        W2W_1_1_4_2_1_1_1_1 : WSTRING2WSTRING(IN := %opcuaGoodRemoteWrite%);
        W2W_1_1_4_2_1_1_1_1_1 : WSTRING2WSTRING(IN := %opcuaGoodCreateMethod1%);
        W2W_1_1_4_2_1_1_1_1_1_1 : WSTRING2WSTRING(IN := %opcuaGoodCallMethod1%);
        W2W_1_1_4_2_1_1_1_1_1_1_1 : WSTRING2WSTRING(IN := %opcuaGoodSubscribe1%);
        W2W_2 : WSTRING2WSTRING(IN := %opcuaGUIDIdentifier%);
      END_FBS
      SUBAPPLICATION NoSemicolon
        EVENT_INPUT
          REQ;
        END_EVENT
        EVENT_OUTPUT
          CNF;
        END_EVENT
        VAR_INPUT
          ID : ANY_ELEMENTARY;
        END_VAR
      END_SUBAPPLICATION
      SUBAPPLICATION emptyAction
        EVENT_INPUT
          REQ;
        END_EVENT
        EVENT_OUTPUT
          CNF;
        END_EVENT
        VAR_INPUT
          ID : WSTRING;
        END_VAR
      END_SUBAPPLICATION
      SUBAPPLICATION NoExistingAction
        EVENT_INPUT
          REQ;
        END_EVENT
        EVENT_OUTPUT
          CNF;
        END_EVENT
        VAR_INPUT
          ID : WSTRING;
        END_VAR
      END_SUBAPPLICATION
      SUBAPPLICATION UnknownIdentifier
        EVENT_INPUT
          REQ;
        END_EVENT
        EVENT_OUTPUT
          CNF;
        END_EVENT
        VAR_INPUT
          ID : WSTRING;
        END_VAR
      END_SUBAPPLICATION
      SUBAPPLICATION WrongIdentifier
        EVENT_INPUT
          REQ;
        END_EVENT
        EVENT_OUTPUT
          CNF;
        END_EVENT
        VAR_INPUT
          ID : WSTRING;
        END_VAR
      END_SUBAPPLICATION
      SUBAPPLICATION wrongNodeId
        EVENT_INPUT
          REQ;
        END_EVENT
        EVENT_OUTPUT
          CNF;
        END_EVENT
        VAR_INPUT
          ID : WSTRING;
        END_VAR
      END_SUBAPPLICATION
      SUBAPPLICATION wrongPair
        EVENT_INPUT
          REQ;
        END_EVENT
        EVENT_OUTPUT
          CNF;
        END_EVENT
        VAR_INPUT
          ID : WSTRING;
        END_VAR
      END_SUBAPPLICATION
      SUBAPPLICATION LocalWithoutBrowseName
        EVENT_INPUT
          REQ;
        END_EVENT
        EVENT_OUTPUT
          CNF;
        END_EVENT
        VAR_INPUT
          ID : WSTRING;
        END_VAR
      END_SUBAPPLICATION
      SUBAPPLICATION RemoteWithoutBrowseNameNorNodeId
        EVENT_INPUT
          REQ;
        END_EVENT
        EVENT_OUTPUT
          CNF;
        END_EVENT
        VAR_INPUT
          ID : WSTRING;
        END_VAR
      END_SUBAPPLICATION
      SUBAPPLICATION RemoteRead
        EVENT_INPUT
          REQ;
        END_EVENT
        EVENT_OUTPUT
          CNF;
        END_EVENT
        VAR_INPUT
          ID : WSTRING;
        END_VAR
      END_SUBAPPLICATION
      SUBAPPLICATION LocalRead
        EVENT_INPUT
          REQ;
        END_EVENT
        EVENT_OUTPUT
          CNF;
        END_EVENT
        VAR_INPUT
          ID : WSTRING;
        END_VAR
      END_SUBAPPLICATION
      SUBAPPLICATION RemoteWrite
        EVENT_INPUT
          REQ;
        END_EVENT
        EVENT_OUTPUT
          CNF;
        END_EVENT
        VAR_INPUT
          ID : WSTRING;
        END_VAR
      END_SUBAPPLICATION
      SUBAPPLICATION LocalWrite
        EVENT_INPUT
          REQ;
        END_EVENT
        EVENT_OUTPUT
          CNF;
        END_EVENT
        VAR_INPUT
          ID : WSTRING;
        END_VAR
      END_SUBAPPLICATION
      SUBAPPLICATION CreateMethod
        EVENT_INPUT
          REQ;
        END_EVENT
        EVENT_OUTPUT
          CNF;
        END_EVENT
        VAR_INPUT
          ID : WSTRING;
        END_VAR
      END_SUBAPPLICATION
      SUBAPPLICATION CallMethod
        EVENT_INPUT
          REQ;
        END_EVENT
        EVENT_OUTPUT
          CNF;
        END_EVENT
        VAR_INPUT
          ID : WSTRING;
        END_VAR
      END_SUBAPPLICATION
      SUBAPPLICATION Subscribe
        EVENT_INPUT
          REQ;
        END_EVENT
        EVENT_OUTPUT
          CNF;
        END_EVENT
        VAR_INPUT
          ID : WSTRING;
        END_VAR
      END_SUBAPPLICATION
      SUBAPPLICATION GUIDIdentifier
        EVENT_INPUT
          REQ;
        END_EVENT
        EVENT_OUTPUT
          CNF;
        END_EVENT
        VAR_INPUT
          ID : WSTRING;
        END_VAR
      END_SUBAPPLICATION
      EVENT_CONNECTIONS
        NoSemicolon.CNF TO W2W_1.REQ;
        W2W_1.CNF TO emptyAction.REQ;
        emptyAction.CNF TO W2W_1_1.REQ;
        W2W_1_1.CNF TO NoExistingAction.REQ;
        NoExistingAction.CNF TO W2W_1_1_1.REQ;
        UnknownIdentifier.CNF TO W2W_1_1_4.REQ;
        W2W_1_1_4.CNF TO WrongIdentifier.REQ;
        W2W_1_1_3.CNF TO UnknownIdentifier.REQ;
        W2W_1_1_2.CNF TO wrongNodeId.REQ;
        wrongNodeId.CNF TO W2W_1_1_3.REQ;
        W2W_1_1_1.CNF TO wrongPair.REQ;
        wrongPair.CNF TO W2W_1_1_2.REQ;
        W2W.CNF TO NoSemicolon.REQ;
        WrongIdentifier.CNF TO W2W_1_1_4_1.REQ;
        W2W_1_1_4_1.CNF TO LocalWithoutBrowseName.REQ;
        LocalWithoutBrowseName.CNF TO W2W_1_1_4_2.REQ;
        W2W_1_1_4_2.CNF TO RemoteWithoutBrowseNameNorNodeId.REQ;
        W2W_1_1_4_2_1_1.CNF TO RemoteRead.REQ;
        LocalRead.CNF TO W2W_1_1_4_2_1_1.REQ;
        RemoteWithoutBrowseNameNorNodeId.CNF TO W2W_1_1_4_2_1.REQ;
        W2W_1_1_4_2_1.CNF TO LocalRead.REQ;
        RemoteRead.CNF TO W2W_1_1_4_2_1_1_1.REQ;
        W2W_1_1_4_2_1_1_1_1.CNF TO RemoteWrite.REQ;
        W2W_1_1_4_2_1_1_1.CNF TO LocalWrite.REQ;
        LocalWrite.CNF TO W2W_1_1_4_2_1_1_1_1.REQ;
        W2W_1_1_4_2_1_1_1_1_1.CNF TO CreateMethod.REQ;
        RemoteWrite.CNF TO W2W_1_1_4_2_1_1_1_1_1.REQ;
        CreateMethod.CNF TO W2W_1_1_4_2_1_1_1_1_1_1.REQ;
        W2W_1_1_4_2_1_1_1_1_1_1.CNF TO CallMethod.REQ;
        Subscribe.CNF TO STEST_END.REQ;
        CallMethod.CNF TO W2W_1_1_4_2_1_1_1_1_1_1_1.REQ;
        W2W_1_1_4_2_1_1_1_1_1_1_1.CNF TO Subscribe.REQ;
        W2W_2.CNF TO GUIDIdentifier.REQ;
        GUIDIdentifier.CNF TO W2W.REQ;
        START.WARM TO W2W_2.REQ;
        START.COLD TO W2W_2.REQ;
      END_CONNECTIONS
      DATA_CONNECTIONS
        W2W_1_1_4.OUT TO WrongIdentifier.ID;
        W2W_1_1_3.OUT TO UnknownIdentifier.ID;
        W2W_1_1_2.OUT TO wrongNodeId.ID;
        W2W_1_1_1.OUT TO wrongPair.ID;
        W2W_1_1.OUT TO NoExistingAction.ID;
        W2W_1.OUT TO emptyAction.ID;
        W2W.OUT TO NoSemicolon.ID;
        W2W_1_1_4_1.OUT TO LocalWithoutBrowseName.ID;
        W2W_1_1_4_2.OUT TO RemoteWithoutBrowseNameNorNodeId.ID;
        W2W_1_1_4_2_1_1.OUT TO RemoteRead.ID;
        W2W_1_1_4_2_1.OUT TO LocalRead.ID;
        W2W_1_1_4_2_1_1_1_1.OUT TO RemoteWrite.ID;
        W2W_1_1_4_2_1_1_1.OUT TO LocalWrite.ID;
        W2W_1_1_4_2_1_1_1_1_1.OUT TO CreateMethod.ID;
        W2W_1_1_4_2_1_1_1_1_1_1.OUT TO CallMethod.ID;
        W2W_1_1_4_2_1_1_1_1_1_1_1.OUT TO Subscribe.ID;
        W2W_2.OUT TO GUIDIdentifier.ID;
      END_CONNECTIONS
    END_RESOURCE
    RESOURCE foldersReadFirst : EMB_RES
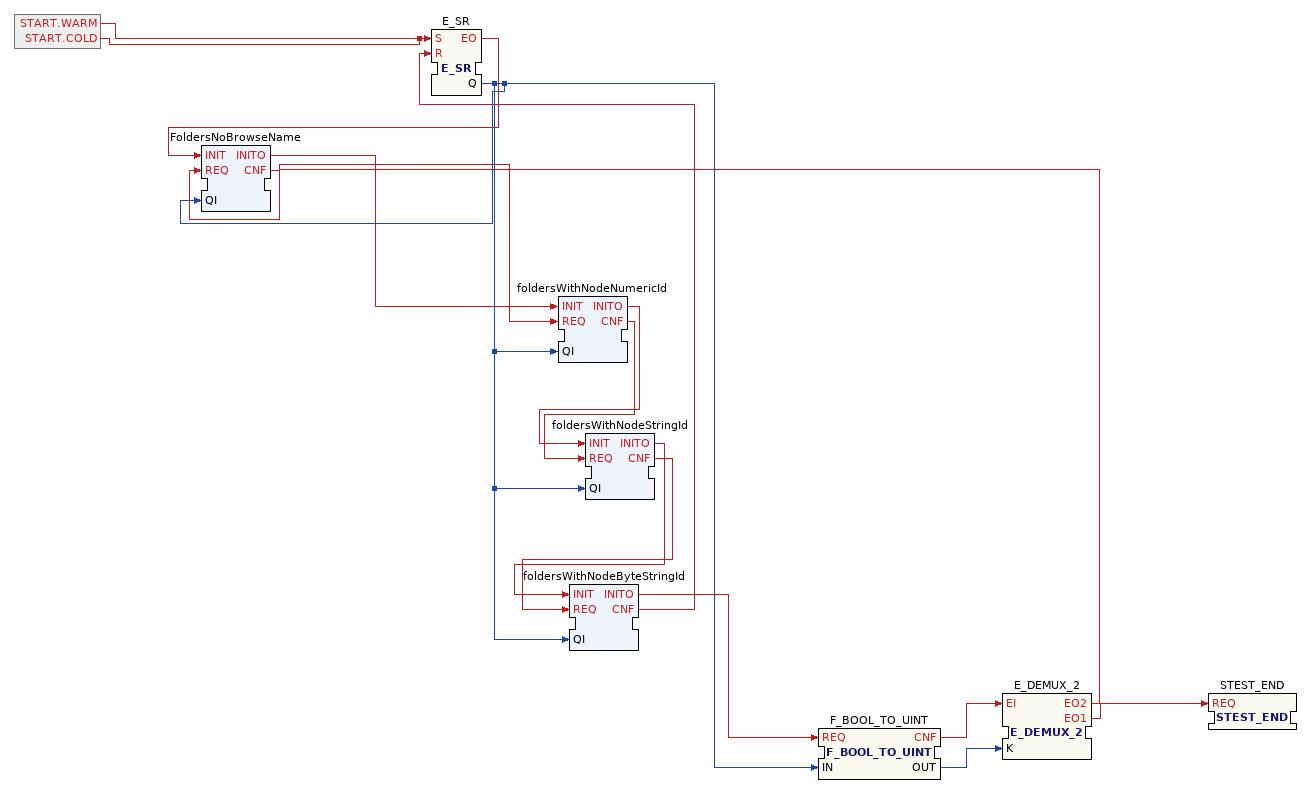
      FBS
        E_SR : E_SR;
        STEST_END : STEST_END;
        E_DEMUX_2 : E_DEMUX_2;
        F_BOOL_TO_UINT : F_BOOL_TO_UINT;
      END_FBS
      SUBAPPLICATION FoldersNoBrowseName
        EVENT_INPUT
          INIT;
          REQ;
        END_EVENT
        EVENT_OUTPUT
          INITO;
          CNF;
        END_EVENT
        VAR_INPUT
          QI : BOOL;
        END_VAR
      END_SUBAPPLICATION
      SUBAPPLICATION foldersWithNodeStringId
        EVENT_INPUT
          INIT;
          REQ;
        END_EVENT
        EVENT_OUTPUT
          INITO;
          CNF;
        END_EVENT
        VAR_INPUT
          QI : BOOL;
        END_VAR
      END_SUBAPPLICATION
      SUBAPPLICATION foldersWithNodeNumericId
        EVENT_INPUT
          INIT;
          REQ;
        END_EVENT
        EVENT_OUTPUT
          INITO;
          CNF;
        END_EVENT
        VAR_INPUT
          QI : BOOL;
        END_VAR
      END_SUBAPPLICATION
      SUBAPPLICATION foldersWithNodeByteStringId
        EVENT_INPUT
          INIT;
          REQ;
        END_EVENT
        EVENT_OUTPUT
          INITO;
          CNF;
        END_EVENT
        VAR_INPUT
          QI : BOOL;
        END_VAR
      END_SUBAPPLICATION
      EVENT_CONNECTIONS
        START.WARM TO E_SR.S;
        START.COLD TO E_SR.S;
        E_SR.EO TO FoldersNoBrowseName.INIT;
        foldersWithNodeStringId.INITO TO foldersWithNodeByteStringId.INIT;
        foldersWithNodeStringId.CNF TO foldersWithNodeByteStringId.REQ;
        E_DEMUX_2.EO2 TO FoldersNoBrowseName.REQ;
        F_BOOL_TO_UINT.CNF TO E_DEMUX_2.EI;
        foldersWithNodeByteStringId.INITO TO F_BOOL_TO_UINT.REQ;
        foldersWithNodeNumericId.CNF TO foldersWithNodeStringId.REQ;
        foldersWithNodeByteStringId.CNF TO E_SR.R;
        foldersWithNodeNumericId.INITO TO foldersWithNodeStringId.INIT;
        FoldersNoBrowseName.INITO TO foldersWithNodeNumericId.INIT;
        FoldersNoBrowseName.CNF TO foldersWithNodeNumericId.REQ;
        E_DEMUX_2.EO1 TO STEST_END.REQ;
      END_CONNECTIONS
      DATA_CONNECTIONS
        E_SR.Q TO FoldersNoBrowseName.QI;
        E_SR.Q TO foldersWithNodeStringId.QI;
        E_SR.Q TO foldersWithNodeNumericId.QI;
        E_SR.Q TO foldersWithNodeByteStringId.QI;
        E_SR.Q TO F_BOOL_TO_UINT.IN;
        F_BOOL_TO_UINT.OUT TO E_DEMUX_2.K;
      END_CONNECTIONS
    END_RESOURCE
    RESOURCE foldersWriteFirst : EMB_RES
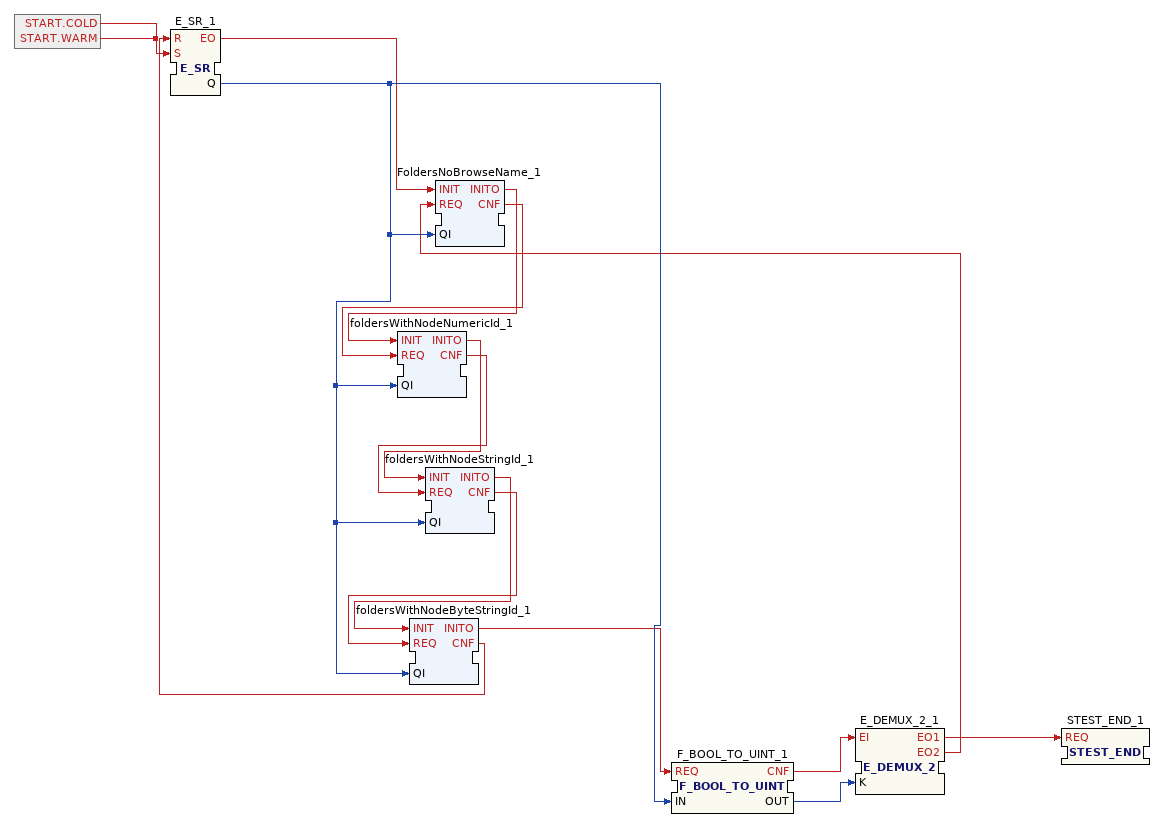
      FBS
        STEST_END_1 : STEST_END;
        F_BOOL_TO_UINT_1 : F_BOOL_TO_UINT;
        E_DEMUX_2_1 : E_DEMUX_2;
        E_SR_1 : E_SR;
      END_FBS
      SUBAPPLICATION FoldersNoBrowseName_1
        EVENT_INPUT
          INIT;
          REQ;
        END_EVENT
        EVENT_OUTPUT
          INITO;
          CNF;
        END_EVENT
        VAR_INPUT
          QI : BOOL;
        END_VAR
      END_SUBAPPLICATION
      SUBAPPLICATION foldersWithNodeByteStringId_1
        EVENT_INPUT
          INIT;
          REQ;
        END_EVENT
        EVENT_OUTPUT
          INITO;
          CNF;
        END_EVENT
        VAR_INPUT
          QI : BOOL;
        END_VAR
      END_SUBAPPLICATION
      SUBAPPLICATION foldersWithNodeNumericId_1
        EVENT_INPUT
          INIT;
          REQ;
        END_EVENT
        EVENT_OUTPUT
          INITO;
          CNF;
        END_EVENT
        VAR_INPUT
          QI : BOOL;
        END_VAR
      END_SUBAPPLICATION
      SUBAPPLICATION foldersWithNodeStringId_1
        EVENT_INPUT
          INIT;
          REQ;
        END_EVENT
        EVENT_OUTPUT
          INITO;
          CNF;
        END_EVENT
        VAR_INPUT
          QI : BOOL;
        END_VAR
      END_SUBAPPLICATION
      EVENT_CONNECTIONS
        FoldersNoBrowseName_1.INITO TO foldersWithNodeNumericId_1.INIT;
        FoldersNoBrowseName_1.CNF TO foldersWithNodeNumericId_1.REQ;
        foldersWithNodeByteStringId_1.INITO TO F_BOOL_TO_UINT_1.REQ;
        foldersWithNodeNumericId_1.INITO TO foldersWithNodeStringId_1.INIT;
        foldersWithNodeNumericId_1.CNF TO foldersWithNodeStringId_1.REQ;
        foldersWithNodeStringId_1.INITO TO foldersWithNodeByteStringId_1.INIT;
        foldersWithNodeStringId_1.CNF TO foldersWithNodeByteStringId_1.REQ;
        F_BOOL_TO_UINT_1.CNF TO E_DEMUX_2_1.EI;
        E_DEMUX_2_1.EO1 TO STEST_END_1.REQ;
        E_DEMUX_2_1.EO2 TO FoldersNoBrowseName_1.REQ;
        foldersWithNodeByteStringId_1.CNF TO E_SR_1.R;
        E_SR_1.EO TO FoldersNoBrowseName_1.INIT;
        START.COLD TO E_SR_1.S;
        START.WARM TO E_SR_1.S;
      END_CONNECTIONS
      DATA_CONNECTIONS
        F_BOOL_TO_UINT_1.OUT TO E_DEMUX_2_1.K;
        E_SR_1.Q TO foldersWithNodeStringId_1.QI;
        E_SR_1.Q TO foldersWithNodeNumericId_1.QI;
        E_SR_1.Q TO FoldersNoBrowseName_1.QI;
        E_SR_1.Q TO foldersWithNodeByteStringId_1.QI;
        E_SR_1.Q TO F_BOOL_TO_UINT_1.IN;
      END_CONNECTIONS
    END_RESOURCE
    RESOURCE createLocalMethods : EMB_RES
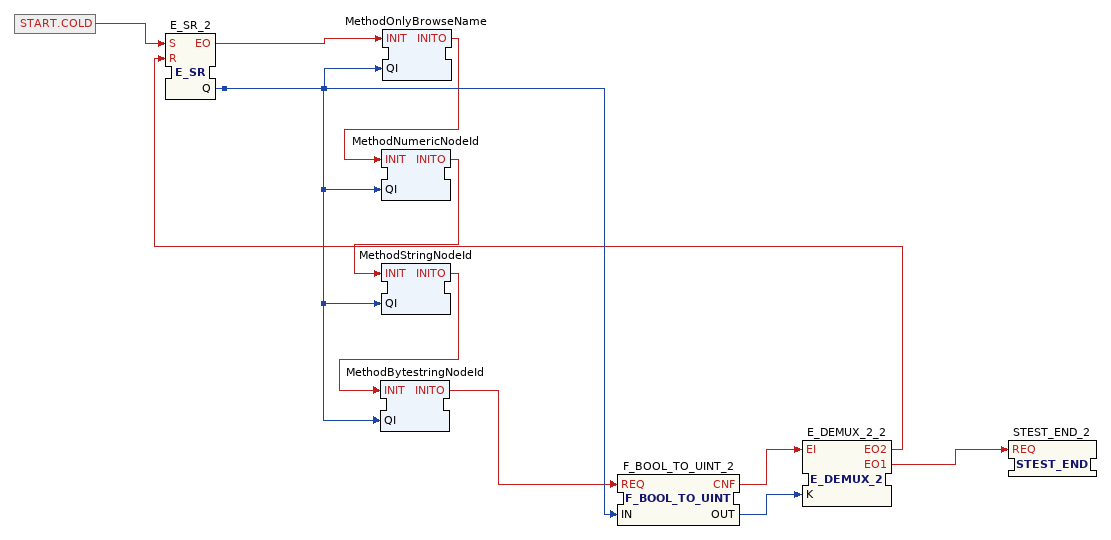
      FBS
        F_BOOL_TO_UINT_2 : F_BOOL_TO_UINT;
        E_DEMUX_2_2 : E_DEMUX_2;
        E_SR_2 : E_SR;
        STEST_END_2 : STEST_END;
      END_FBS
      SUBAPPLICATION MethodOnlyBrowseName
        EVENT_INPUT
          INIT;
        END_EVENT
        EVENT_OUTPUT
          INITO;
        END_EVENT
        VAR_INPUT
          QI : BOOL;
        END_VAR
      END_SUBAPPLICATION
      SUBAPPLICATION MethodBytestringNodeId
        EVENT_INPUT
          INIT;
        END_EVENT
        EVENT_OUTPUT
          INITO;
        END_EVENT
        VAR_INPUT
          QI : BOOL;
        END_VAR
      END_SUBAPPLICATION
      SUBAPPLICATION MethodNumericNodeId
        EVENT_INPUT
          INIT;
        END_EVENT
        EVENT_OUTPUT
          INITO;
        END_EVENT
        VAR_INPUT
          QI : BOOL;
        END_VAR
      END_SUBAPPLICATION
      SUBAPPLICATION MethodStringNodeId
        EVENT_INPUT
          INIT;
        END_EVENT
        EVENT_OUTPUT
          INITO;
        END_EVENT
        VAR_INPUT
          QI : BOOL;
        END_VAR
      END_SUBAPPLICATION
      EVENT_CONNECTIONS
        F_BOOL_TO_UINT_2.CNF TO E_DEMUX_2_2.EI;
        E_SR_2.EO TO MethodOnlyBrowseName.INIT;
        MethodOnlyBrowseName.INITO TO MethodNumericNodeId.INIT;
        MethodNumericNodeId.INITO TO MethodStringNodeId.INIT;
        MethodStringNodeId.INITO TO MethodBytestringNodeId.INIT;
        START.COLD TO E_SR_2.S;
        E_DEMUX_2_2.EO2 TO E_SR_2.R;
        E_DEMUX_2_2.EO1 TO STEST_END_2.REQ;
        MethodBytestringNodeId.INITO TO F_BOOL_TO_UINT_2.REQ;
      END_CONNECTIONS
      DATA_CONNECTIONS
        F_BOOL_TO_UINT_2.OUT TO E_DEMUX_2_2.K;
        E_SR_2.Q TO MethodOnlyBrowseName.QI;
        E_SR_2.Q TO MethodBytestringNodeId.QI;
        E_SR_2.Q TO F_BOOL_TO_UINT_2.IN;
        E_SR_2.Q TO MethodNumericNodeId.QI;
        E_SR_2.Q TO MethodStringNodeId.QI;
      END_CONNECTIONS
    END_RESOURCE
    RESOURCE WorkingServer : EMB_RES
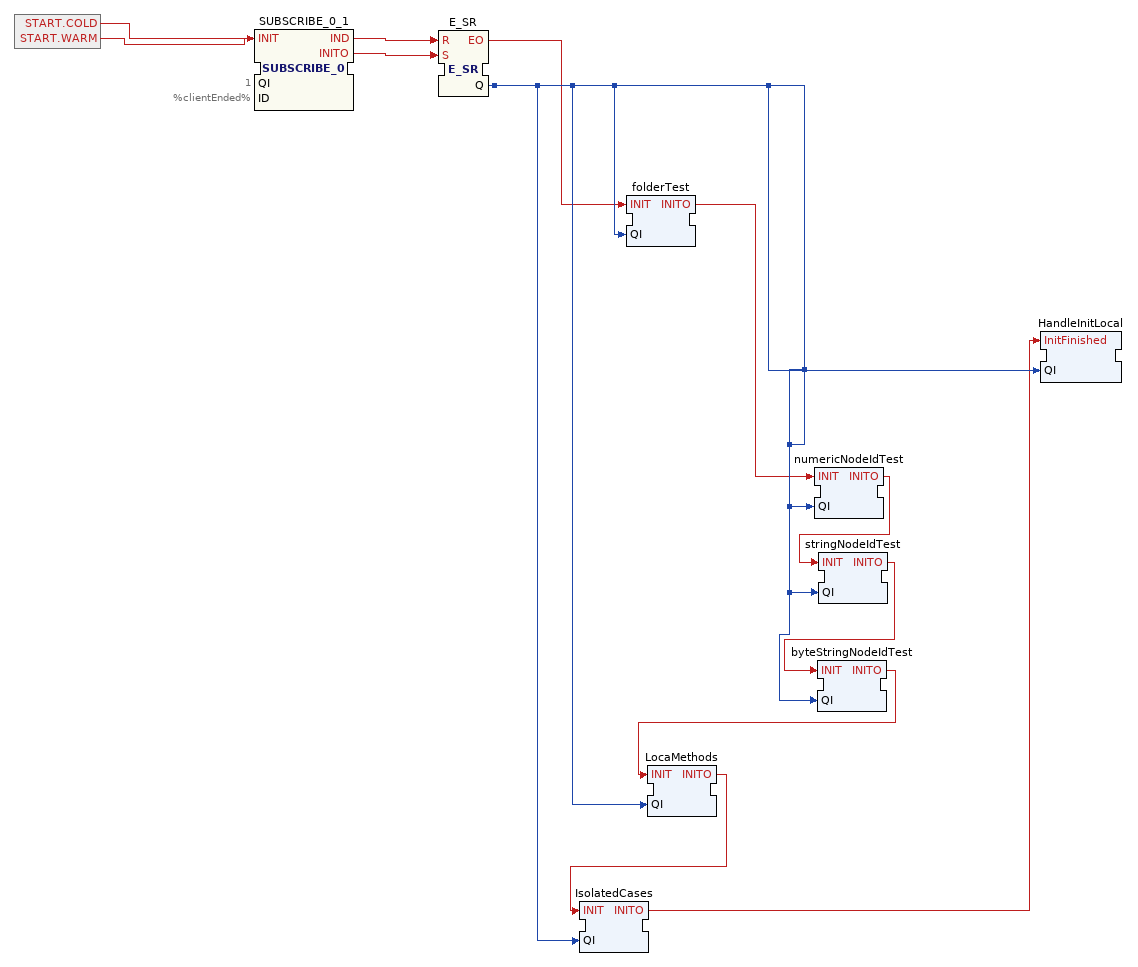
      FBS
        E_SR : E_SR;
        SUBSCRIBE_0_1 : SUBSCRIBE_0(QI := 1, ID := %clientEnded%);
      END_FBS
      SUBAPPLICATION folderTest
        EVENT_INPUT
          INIT;
        END_EVENT
        EVENT_OUTPUT
          INITO;
        END_EVENT
        VAR_INPUT
          QI : BOOL;
        END_VAR
      END_SUBAPPLICATION
      SUBAPPLICATION HandleInitLocal
        EVENT_INPUT
          InitFinished;
        END_EVENT
        VAR_INPUT
          QI : BOOL;
        END_VAR
      END_SUBAPPLICATION
      SUBAPPLICATION LocaMethods
        EVENT_INPUT
          INIT;
        END_EVENT
        EVENT_OUTPUT
          INITO;
        END_EVENT
        VAR_INPUT
          QI : BOOL;
        END_VAR
      END_SUBAPPLICATION
      SUBAPPLICATION stringNodeIdTest
        EVENT_INPUT
          INIT;
        END_EVENT
        EVENT_OUTPUT
          INITO;
        END_EVENT
        VAR_INPUT
          QI : BOOL;
        END_VAR
      END_SUBAPPLICATION
      SUBAPPLICATION byteStringNodeIdTest
        EVENT_INPUT
          INIT;
        END_EVENT
        EVENT_OUTPUT
          INITO;
        END_EVENT
        VAR_INPUT
          QI : BOOL;
        END_VAR
      END_SUBAPPLICATION
      SUBAPPLICATION numericNodeIdTest
        EVENT_INPUT
          INIT;
        END_EVENT
        EVENT_OUTPUT
          INITO;
        END_EVENT
        VAR_INPUT
          QI : BOOL;
        END_VAR
      END_SUBAPPLICATION
      SUBAPPLICATION IsolatedCases
        EVENT_INPUT
          INIT;
        END_EVENT
        EVENT_OUTPUT
          INITO;
        END_EVENT
        VAR_INPUT
          QI : BOOL;
        END_VAR
      END_SUBAPPLICATION
      EVENT_CONNECTIONS
        SUBSCRIBE_0_1.IND TO E_SR.R;
        SUBSCRIBE_0_1.INITO TO E_SR.S;
        START.COLD TO SUBSCRIBE_0_1.INIT;
        START.WARM TO SUBSCRIBE_0_1.INIT;
        E_SR.EO TO folderTest.INIT;
        numericNodeIdTest.INITO TO stringNodeIdTest.INIT;
        stringNodeIdTest.INITO TO byteStringNodeIdTest.INIT;
        byteStringNodeIdTest.INITO TO LocaMethods.INIT;
        folderTest.INITO TO numericNodeIdTest.INIT;
        LocaMethods.INITO TO IsolatedCases.INIT;
        IsolatedCases.INITO TO HandleInitLocal.InitFinished;
      END_CONNECTIONS
      DATA_CONNECTIONS
        E_SR.Q TO folderTest.QI;
        E_SR.Q TO HandleInitLocal.QI;
        E_SR.Q TO numericNodeIdTest.QI;
        E_SR.Q TO stringNodeIdTest.QI;
        E_SR.Q TO byteStringNodeIdTest.QI;
        E_SR.Q TO LocaMethods.QI;
        E_SR.Q TO IsolatedCases.QI;
      END_CONNECTIONS
    END_RESOURCE
    RESOURCE FailingServer : EMB_RES
      FBS
        E_SWITCH : E_SWITCH;
        WorngInputs : TEST_CONDITION(check := 0);
        E_SR : E_SR;
        GoodInputs : TEST_CONDITION;
        SUBSCRIBE_0_1 : SUBSCRIBE_0(QI := 1, ID := %clientEnded%);
        WorngInputsOutputs : TEST_CONDITION(check := 0);
        Writable1 : PUBLISH_1(QI := 1, ID := opc_ua[WRITE;%opcuaFolderTestWithNodeIdNumeric1%/]);
        WorngInputsType : TEST_CONDITION(check := 0);
        BOOL2BOOL_2_1 : DINT2DINT(IN := %opcuaReadValue1%);
        SERVER_0 : SERVER_1(QI := 1, ID := opc_ua[%localMethodAction%;%opcuaMethodCreation5%]);
        SERVER_0_1 : SERVER_1(QI := 1, ID := opc_ua[%localMethodAction%;%opcuaMethodCreation6%]);
        SERVER_0_1_1 : SERVER_1(QI := 1, ID := opc_ua[%localMethodAction%;%opcuaMethodCreation7%]);
        DINT2DINT : DINT2DINT;
        DINT2DINT_1_1 : DINT2DINT;
        DINT2DINT_1 : DINT2DINT;
        SameNodeIdWrite : TEST_CONDITION;
        BOOL2BOOL_2_1_1 : DINT2DINT(IN := %opcuaReadValue1%);
        Writable1_1 : PUBLISH_1(QI := 1, ID := opc_ua[WRITE;/Objects/firstRead/NumericNodeId/folderTests/WithId1,1:i=12345]);
        BOOL2BOOL_2_1_1_1 : DINT2DINT(IN := %opcuaReadValue1%);
        SameNameDifferentNodeIdW : TEST_CONDITION;
        Writable1_1_1 : PUBLISH_1(QI := 1, ID := opc_ua[WRITE;/Objects/firstRead/StringNodeId/folderTests/WithId,1:s=helloWrite]);
        SUBSCRIBE_1_1 : SUBSCRIBE_1(QI := 1, ID := opc_ua[READ;%opcuaFolderTestWithNodeIdNumeric1%]);
        BOOL2BOOL_3_1 : DINT2DINT;
        SUBSCRIBE_1_1_1 : SUBSCRIBE_1(QI := 1, ID := opc_ua[READ;%opcuaFolderTestWithNodeIdNumeric1%]);
        BOOL2BOOL_3 : DINT2DINT;
        SameNodeSecondRead : TEST_CONDITION;
        ReadExistingWritable : TEST_CONDITION;
        F_NOT_1_1 : F_NOT;
        F_NOT : F_NOT;
        SUBSCRIBE_1_1_1_1 : SUBSCRIBE_1(QI := 1, ID := opc_ua[READ;/Objects/firstRead/StringNodeId/folderTests/WithId,1:s=hello]);
        SUBSCRIBE_wrongPath : SUBSCRIBE_1(QI := 1, ID := opc_ua[READ;///]);
        F_NOT_1_2_1_1 : F_NOT;
        SERVER_0_2 : SERVER_1(QI := 1, ID := opc_ua[%localMethodAction%;%opcuaMethodCreation5%]);
        DoubleMethod : TEST_CONDITION;
        BOOL2BOOL_3_2 : DINT2DINT;
        BOOL2BOOL_3_1_1_1 : DINT2DINT;
        F_NOT_1_2_1 : F_NOT;
        ValidNode : TEST_CONDITION;
        WrongPath : TEST_CONDITION;
        BOOL2BOOL_3_1_1 : DINT2DINT;
        BOOL2BOOL_3_2_1_1 : DINT2DINT;
        F_NOT_1_2_1_1_1_1 : F_NOT;
        SUBSCRIBE_150 : SUBSCRIBE_1(QI := 1, ID := opc_ua[READ;%opcuaFolderTestWithNodeIdByteString1%]);
        UnconnectedRD : TEST_CONDITION;
        UnconnectedSD : TEST_CONDITION;
        BOOL2BOOL_3_2_1 : DINT2DINT;
        STRING2STRING_1 : STRING2STRING;
        F_NOT_1 : F_NOT;
        F_NOT_1_2_1_1_1 : F_NOT;
        DifferentTypesOutput : TEST_CONDITION;
        SUBSCRIBE_140 : SUBSCRIBE_2(QI := 1, ID := opc_ua[READ;%opcuaFolderTestWithNodeIdString1%;%opcuaFolderTestWithNodeIdByteString2%]);
        Writable1_1_2 : PUBLISH_2(QI := 1, ID := opc_ua[WRITE;%opcuaFolderTestWithNodeIdString1%;%opcuaFolderTestWithNodeIdByteString2%]);
        SameNodeIdRead : TEST_CONDITION;
        SUBSCRIBE_1 : SUBSCRIBE_1(QI := 1, ID := opc_ua[READ;/Objects/firstRead/NumericNodeId/folderTests/WithId1,1:i=12345]);
        BOOL2BOOL_2_1_1_2 : DINT2DINT;
        F_NOT_2 : F_NOT;
        F_EQ : F_EQ(IN2 := %opcuaReadValue1%);
        SameNameDifferentNodeIdR : TEST_CONDITION;
        Writable1_2 : SUBSCRIBE_1(QI := 1, ID := opc_ua[READ;/Objects/firstRead/StringNodeId/folderTests/WithId,1:s=helloRead]);
        BOOL2BOOL_3_3 : DINT2DINT;
        STRING2STRING : INT2INT;
        BOOL2BOOL_3_2_1_2 : DINT2DINT;
        SameTypesOutput : TEST_CONDITION;
        SUBSCRIBE_150_1 : SUBSCRIBE_1(QI := 1, ID := opc_ua[READ;/Objects/firstRead/StringNodeId/folderTests/WithId,1:s=hello2]);
        F_NOT_1_2_1_2_1 : F_NOT;
        F_NOT_1_2_1_2 : F_NOT;
        BOOL2BOOL_3_1_1_1_1 : DINT2DINT;
        SUBSCRIBE_NoObject_1 : SUBSCRIBE_1(QI := 1, ID := opc_ua[READ;/Objects/firstRead/Methods/1:1:byteStringNodeId/noOParameters]);
        BOOL2BOOL_3_1_1_1_1_1 : DINT2DINT;
        SUBSCRIBE_NoObject : SUBSCRIBE_1(QI := 1, ID := opc_ua[READ;/firstRead/Methods/byteStringNodeId/noOParameters]);
        BrowseWihtouObject : TEST_CONDITION;
        wrongNamespace1 : TEST_CONDITION;
        STRING2STRING_2 : DINT2DINT;
        Timeoutmethod : SERVER_0(QI := 1, ID := opc_ua[%localMethodAction%;%opcuaMethodCreation8%]);
        E_DELAY_1 : E_DELAY(DT := %methodValidDelay%);
        DINT2DINT_1_2 : DINT2DINT(IN := %opcuaReadValue2%);
        PUBLISH_1 : PUBLISH_1(QI := 1, ID := opc_ua[WRITE;%opcuaWRITEVariable%]);
        SERVER_0_3 : SERVER_0(QI := 1, ID := opc_ua[CREATE_METHOD;/Objects]);
        ObjectsFolder : TEST_CONDITION;
        F_NOT_1_2_1_2_1_1 : F_NOT;
        SERVER_0_4 : SERVER_0(QI := 1, ID := opc_ua[CREATE_METHOD;/Objects/notCalledMethod]);
      END_FBS
      SUBAPPLICATION HandleInitLocal
        EVENT_INPUT
          InitFinished;
        END_EVENT
        VAR_INPUT
          QI : BOOL;
        END_VAR
      END_SUBAPPLICATION
      EVENT_CONNECTIONS
        E_SR.EO TO E_SWITCH.EI;
        SUBSCRIBE_0_1.INITO TO E_SR.S;
        SUBSCRIBE_0_1.IND TO E_SR.R;
        E_SWITCH.EO0 TO HandleInitLocal.InitFinished;
        START.COLD TO SUBSCRIBE_0_1.INIT;
        START.WARM TO SUBSCRIBE_0_1.INIT;
        Writable1.CNF TO WorngInputsType.REQ;
        E_SWITCH.EO1 TO SERVER_0.INIT;
        GoodInputs.CNF TO SERVER_0.RSP;
        SERVER_0.INITO TO SERVER_0_1.INIT;
        WorngInputs.CNF TO SERVER_0_1.RSP;
        SERVER_0_1.IND TO WorngInputs.REQ;
        SERVER_0_1.INITO TO SERVER_0_1_1.INIT;
        WorngInputsOutputs.CNF TO SERVER_0_1_1.RSP;
        SERVER_0_1_1.IND TO WorngInputsOutputs.REQ;
        SUBSCRIBE_1_1.INITO TO ReadExistingWritable.REQ;
        ReadExistingWritable.CNF TO SUBSCRIBE_1_1_1.INIT;
        SUBSCRIBE_1_1_1.INITO TO F_NOT_1_1.REQ;
        F_NOT_1_1.CNF TO SameNodeSecondRead.REQ;
        Writable1_1.INITO TO F_NOT.REQ;
        F_NOT.CNF TO SameNodeIdWrite.REQ;
        SERVER_0_2.INITO TO F_NOT_1_2_1_1.REQ;
        F_NOT_1_2_1_1.CNF TO DoubleMethod.REQ;
        SUBSCRIBE_wrongPath.INITO TO F_NOT_1_2_1.REQ;
        F_NOT_1_2_1.CNF TO WrongPath.REQ;
        Writable1_1_1.INITO TO SameNameDifferentNodeIdW.REQ;
        DoubleMethod.CNF TO SUBSCRIBE_150.INIT;
        F_NOT_1.CNF TO UnconnectedSD.REQ;
        SUBSCRIBE_150.INITO TO F_NOT_1_2_1_1_1.REQ;
        F_NOT_1_2_1_1_1.CNF TO DifferentTypesOutput.REQ;
        F_NOT_1_2_1_1_1_1.CNF TO UnconnectedRD.REQ;
        SUBSCRIBE_140.INITO TO F_NOT_1_2_1_1_1_1.REQ;
        UnconnectedRD.CNF TO Writable1_1_2.INIT;
        Writable1_1_2.INITO TO F_NOT_1.REQ;
        SameNodeIdWrite.CNF TO SUBSCRIBE_1.INIT;
        SUBSCRIBE_1.INITO TO F_NOT_2.REQ;
        F_NOT_2.CNF TO SameNodeIdRead.REQ;
        Writable1.INITO TO Writable1_1.INIT;
        SameNodeSecondRead.CNF TO SERVER_0_2.INIT;
        UnconnectedSD.CNF TO SUBSCRIBE_wrongPath.INIT;
        SameNodeIdRead.CNF TO SUBSCRIBE_1_1_1_1.INIT;
        SUBSCRIBE_1_1_1_1.INITO TO Writable1_2.INIT;
        F_EQ.CNF TO ValidNode.REQ;
        SUBSCRIBE_1_1_1_1.IND TO BOOL2BOOL_3_1_1.REQ;
        BOOL2BOOL_3_1_1.CNF TO F_EQ.REQ;
        Writable1_2.INITO TO SameNameDifferentNodeIdR.REQ;
        SameNameDifferentNodeIdR.CNF TO Writable1_1_1.INIT;
        SameNameDifferentNodeIdW.CNF TO SUBSCRIBE_1_1.INIT;
        SameTypesOutput.CNF TO SUBSCRIBE_140.INIT;
        DifferentTypesOutput.CNF TO SUBSCRIBE_150_1.INIT;
        SUBSCRIBE_150_1.INITO TO SameTypesOutput.REQ;
        WrongPath.CNF TO SUBSCRIBE_NoObject.INIT;
        SUBSCRIBE_NoObject.INITO TO F_NOT_1_2_1_2.REQ;
        F_NOT_1_2_1_2.CNF TO BrowseWihtouObject.REQ;
        BrowseWihtouObject.CNF TO SUBSCRIBE_NoObject_1.INIT;
        F_NOT_1_2_1_2_1.CNF TO wrongNamespace1.REQ;
        SUBSCRIBE_NoObject_1.INITO TO F_NOT_1_2_1_2_1.REQ;
        SERVER_0_1_1.INITO TO Timeoutmethod.INIT;
        Timeoutmethod.INITO TO Writable1.INIT;
        SERVER_0.IND TO E_DELAY_1.START;
        E_DELAY_1.EO TO GoodInputs.REQ;
        wrongNamespace1.CNF TO PUBLISH_1.INIT;
        PUBLISH_1.INITO TO SERVER_0_3.INIT;
        SERVER_0_3.INITO TO F_NOT_1_2_1_2_1_1.REQ;
        F_NOT_1_2_1_2_1_1.CNF TO ObjectsFolder.REQ;
        ObjectsFolder.CNF TO SERVER_0_4.INIT;
        SERVER_0_4.INITO TO SERVER_0_4.RSP;
        SERVER_0_4.INITO TO HandleInitLocal.InitFinished;
      END_CONNECTIONS
      DATA_CONNECTIONS
        E_SR.Q TO E_SWITCH.G;
        BOOL2BOOL_2_1.OUT TO Writable1.SD_1;
        SERVER_0.QO TO GoodInputs.check;
        SERVER_0_1_1.RD_1 TO DINT2DINT.IN;
        DINT2DINT.OUT TO SERVER_0_1_1.SD_1;
        SERVER_0.RD_1 TO DINT2DINT_1_1.IN;
        DINT2DINT_1_1.OUT TO SERVER_0.SD_1;
        SERVER_0_1.RD_1 TO DINT2DINT_1.IN;
        DINT2DINT_1.OUT TO SERVER_0_1.SD_1;
        BOOL2BOOL_2_1_1.OUT TO Writable1_1.SD_1;
        BOOL2BOOL_2_1_1_1.OUT TO Writable1_1_1.SD_1;
        SUBSCRIBE_1_1_1.RD_1 TO BOOL2BOOL_3_1.IN;
        SUBSCRIBE_1_1.RD_1 TO BOOL2BOOL_3.IN;
        SUBSCRIBE_1_1.QO TO ReadExistingWritable.check;
        SUBSCRIBE_1_1_1.QO TO F_NOT_1_1.IN;
        F_NOT_1_1.OUT TO SameNodeSecondRead.check;
        Writable1_1.QO TO F_NOT.IN;
        F_NOT.OUT TO SameNodeIdWrite.check;
        SERVER_0_2.QO TO F_NOT_1_2_1_1.IN;
        F_NOT_1_2_1_1.OUT TO DoubleMethod.check;
        SERVER_0_2.RD_1 TO BOOL2BOOL_3_2.IN;
        BOOL2BOOL_3_2.OUT TO SERVER_0_2.SD_1;
        SUBSCRIBE_wrongPath.RD_1 TO BOOL2BOOL_3_1_1_1.IN;
        SUBSCRIBE_wrongPath.QO TO F_NOT_1_2_1.IN;
        F_NOT_1_2_1.OUT TO WrongPath.check;
        SUBSCRIBE_1_1_1_1.RD_1 TO BOOL2BOOL_3_1_1.IN;
        Writable1_1_1.QO TO SameNameDifferentNodeIdW.check;
        SUBSCRIBE_150.RD_1 TO BOOL2BOOL_3_2_1.IN;
        F_NOT_1.OUT TO UnconnectedSD.check;
        SUBSCRIBE_150.QO TO F_NOT_1_2_1_1_1.IN;
        F_NOT_1_2_1_1_1.OUT TO DifferentTypesOutput.check;
        F_NOT_1_2_1_1_1_1.OUT TO UnconnectedRD.check;
        SUBSCRIBE_140.QO TO F_NOT_1_2_1_1_1_1.IN;
        SUBSCRIBE_140.RD_1 TO BOOL2BOOL_3_2_1_1.IN;
        STRING2STRING_1.OUT TO Writable1_1_2.SD_1;
        Writable1_1_2.QO TO F_NOT_1.IN;
        SUBSCRIBE_1.RD_1 TO BOOL2BOOL_2_1_1_2.IN;
        SUBSCRIBE_1.QO TO F_NOT_2.IN;
        F_NOT_2.OUT TO SameNodeIdRead.check;
        F_EQ.OUT TO ValidNode.check;
        BOOL2BOOL_3_1_1.OUT TO F_EQ.IN1;
        Writable1_2.QO TO SameNameDifferentNodeIdR.check;
        Writable1_2.RD_1 TO BOOL2BOOL_3_3.IN;
        SUBSCRIBE_150.RD_1 TO STRING2STRING.IN;
        E_SR.Q TO HandleInitLocal.QI;
        SUBSCRIBE_150_1.RD_1 TO BOOL2BOOL_3_2_1_2.IN;
        SUBSCRIBE_150_1.QO TO SameTypesOutput.check;
        SUBSCRIBE_NoObject_1.QO TO F_NOT_1_2_1_2_1.IN;
        SUBSCRIBE_NoObject_1.RD_1 TO BOOL2BOOL_3_1_1_1_1_1.IN;
        SUBSCRIBE_NoObject.QO TO F_NOT_1_2_1_2.IN;
        SUBSCRIBE_NoObject.RD_1 TO BOOL2BOOL_3_1_1_1_1.IN;
        F_NOT_1_2_1_2.OUT TO BrowseWihtouObject.check;
        F_NOT_1_2_1_2_1.OUT TO wrongNamespace1.check;
        SUBSCRIBE_150_1.RD_1 TO STRING2STRING_2.IN;
        DINT2DINT_1_2.OUT TO PUBLISH_1.SD_1;
        SERVER_0_3.QO TO F_NOT_1_2_1_2_1_1.IN;
        F_NOT_1_2_1_2_1_1.OUT TO ObjectsFolder.check;
      END_CONNECTIONS
    END_RESOURCE
    RESOURCE delayedWorkingServer : EMB_RES
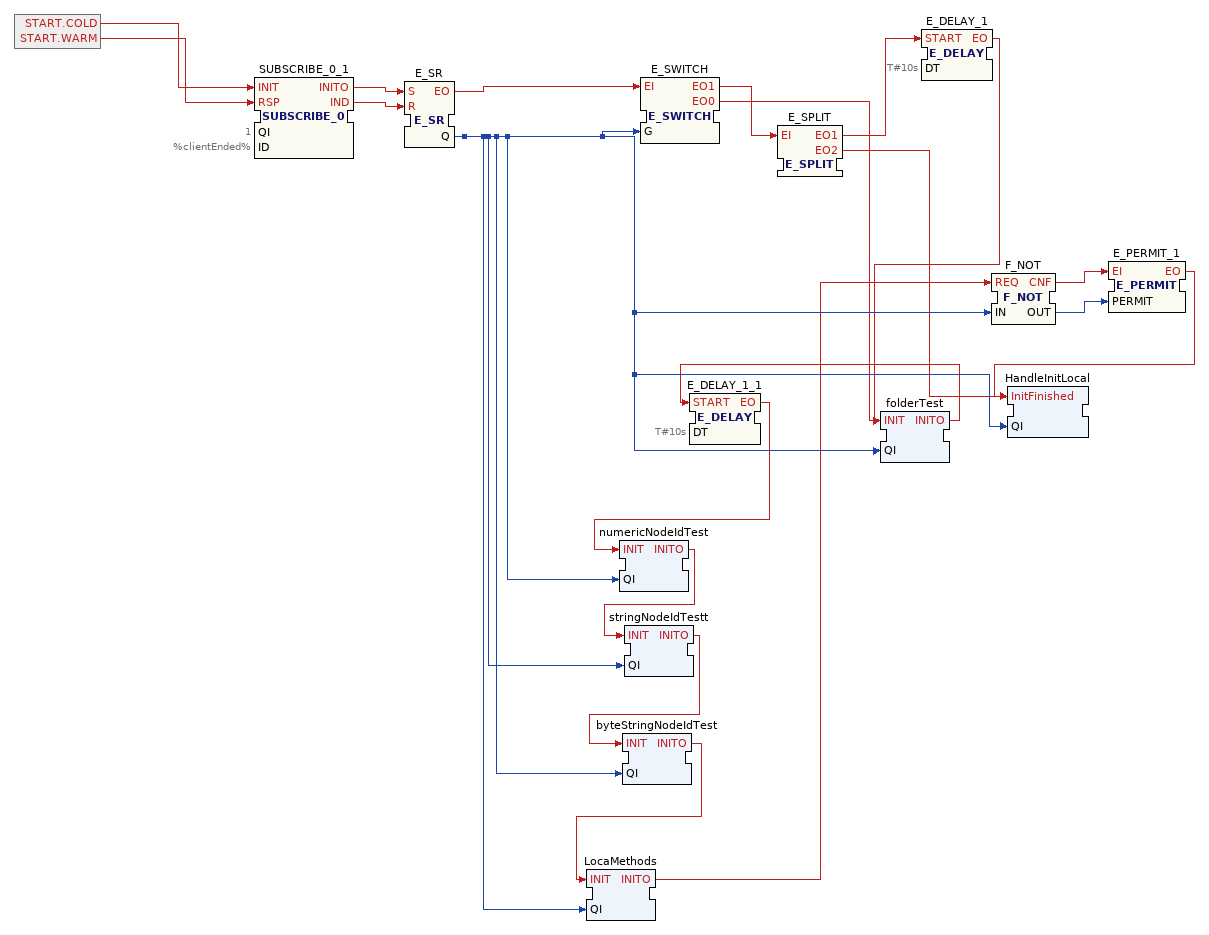
      FBS
        E_SR : E_SR;
        SUBSCRIBE_0_1 : SUBSCRIBE_0(QI := 1, ID := %clientEnded%);
        E_SWITCH : E_SWITCH;
        E_DELAY_1 : E_DELAY(DT := T#10s);
        E_SPLIT : E_SPLIT;
        E_DELAY_1_1 : E_DELAY(DT := T#10s);
        F_NOT : F_NOT;
        E_PERMIT_1 : E_PERMIT;
      END_FBS
      SUBAPPLICATION LocaMethods
        EVENT_INPUT
          INIT;
        END_EVENT
        EVENT_OUTPUT
          INITO;
        END_EVENT
        VAR_INPUT
          QI : BOOL;
        END_VAR
      END_SUBAPPLICATION
      SUBAPPLICATION HandleInitLocal
        EVENT_INPUT
          InitFinished;
        END_EVENT
        VAR_INPUT
          QI : BOOL;
        END_VAR
      END_SUBAPPLICATION
      SUBAPPLICATION numericNodeIdTest
        EVENT_INPUT
          INIT;
        END_EVENT
        EVENT_OUTPUT
          INITO;
        END_EVENT
        VAR_INPUT
          QI : BOOL;
        END_VAR
      END_SUBAPPLICATION
      SUBAPPLICATION folderTest
        EVENT_INPUT
          INIT;
        END_EVENT
        EVENT_OUTPUT
          INITO;
        END_EVENT
        VAR_INPUT
          QI : BOOL;
        END_VAR
      END_SUBAPPLICATION
      SUBAPPLICATION byteStringNodeIdTest
        EVENT_INPUT
          INIT;
        END_EVENT
        EVENT_OUTPUT
          INITO;
        END_EVENT
        VAR_INPUT
          QI : BOOL;
        END_VAR
      END_SUBAPPLICATION
      SUBAPPLICATION stringNodeIdTestt
        EVENT_INPUT
          INIT;
        END_EVENT
        EVENT_OUTPUT
          INITO;
        END_EVENT
        VAR_INPUT
          QI : BOOL;
        END_VAR
      END_SUBAPPLICATION
      EVENT_CONNECTIONS
        SUBSCRIBE_0_1.INITO TO E_SR.S;
        SUBSCRIBE_0_1.IND TO E_SR.R;
        E_SR.EO TO E_SWITCH.EI;
        E_SWITCH.EO1 TO E_SPLIT.EI;
        E_SPLIT.EO1 TO E_DELAY_1.START;
        E_SPLIT.EO2 TO HandleInitLocal.InitFinished;
        LocaMethods.INITO TO F_NOT.REQ;
        F_NOT.CNF TO E_PERMIT_1.EI;
        E_PERMIT_1.EO TO HandleInitLocal.InitFinished;
        START.COLD TO SUBSCRIBE_0_1.INIT;
        START.WARM TO SUBSCRIBE_0_1.RSP;
        numericNodeIdTest.INITO TO stringNodeIdTestt.INIT;
        stringNodeIdTestt.INITO TO byteStringNodeIdTest.INIT;
        folderTest.INITO TO E_DELAY_1_1.START;
        byteStringNodeIdTest.INITO TO LocaMethods.INIT;
        E_SWITCH.EO0 TO folderTest.INIT;
        E_DELAY_1.EO TO folderTest.INIT;
        E_DELAY_1_1.EO TO numericNodeIdTest.INIT;
      END_CONNECTIONS
      DATA_CONNECTIONS
        E_SR.Q TO LocaMethods.QI;
        E_SR.Q TO E_SWITCH.G;
        E_SR.Q TO F_NOT.IN;
        F_NOT.OUT TO E_PERMIT_1.PERMIT;
        E_SR.Q TO HandleInitLocal.QI;
        E_SR.Q TO folderTest.QI;
        E_SR.Q TO stringNodeIdTestt.QI;
        E_SR.Q TO byteStringNodeIdTest.QI;
        E_SR.Q TO numericNodeIdTest.QI;
      END_CONNECTIONS
    END_RESOURCE
    RESOURCE typesServer : EMB_RES
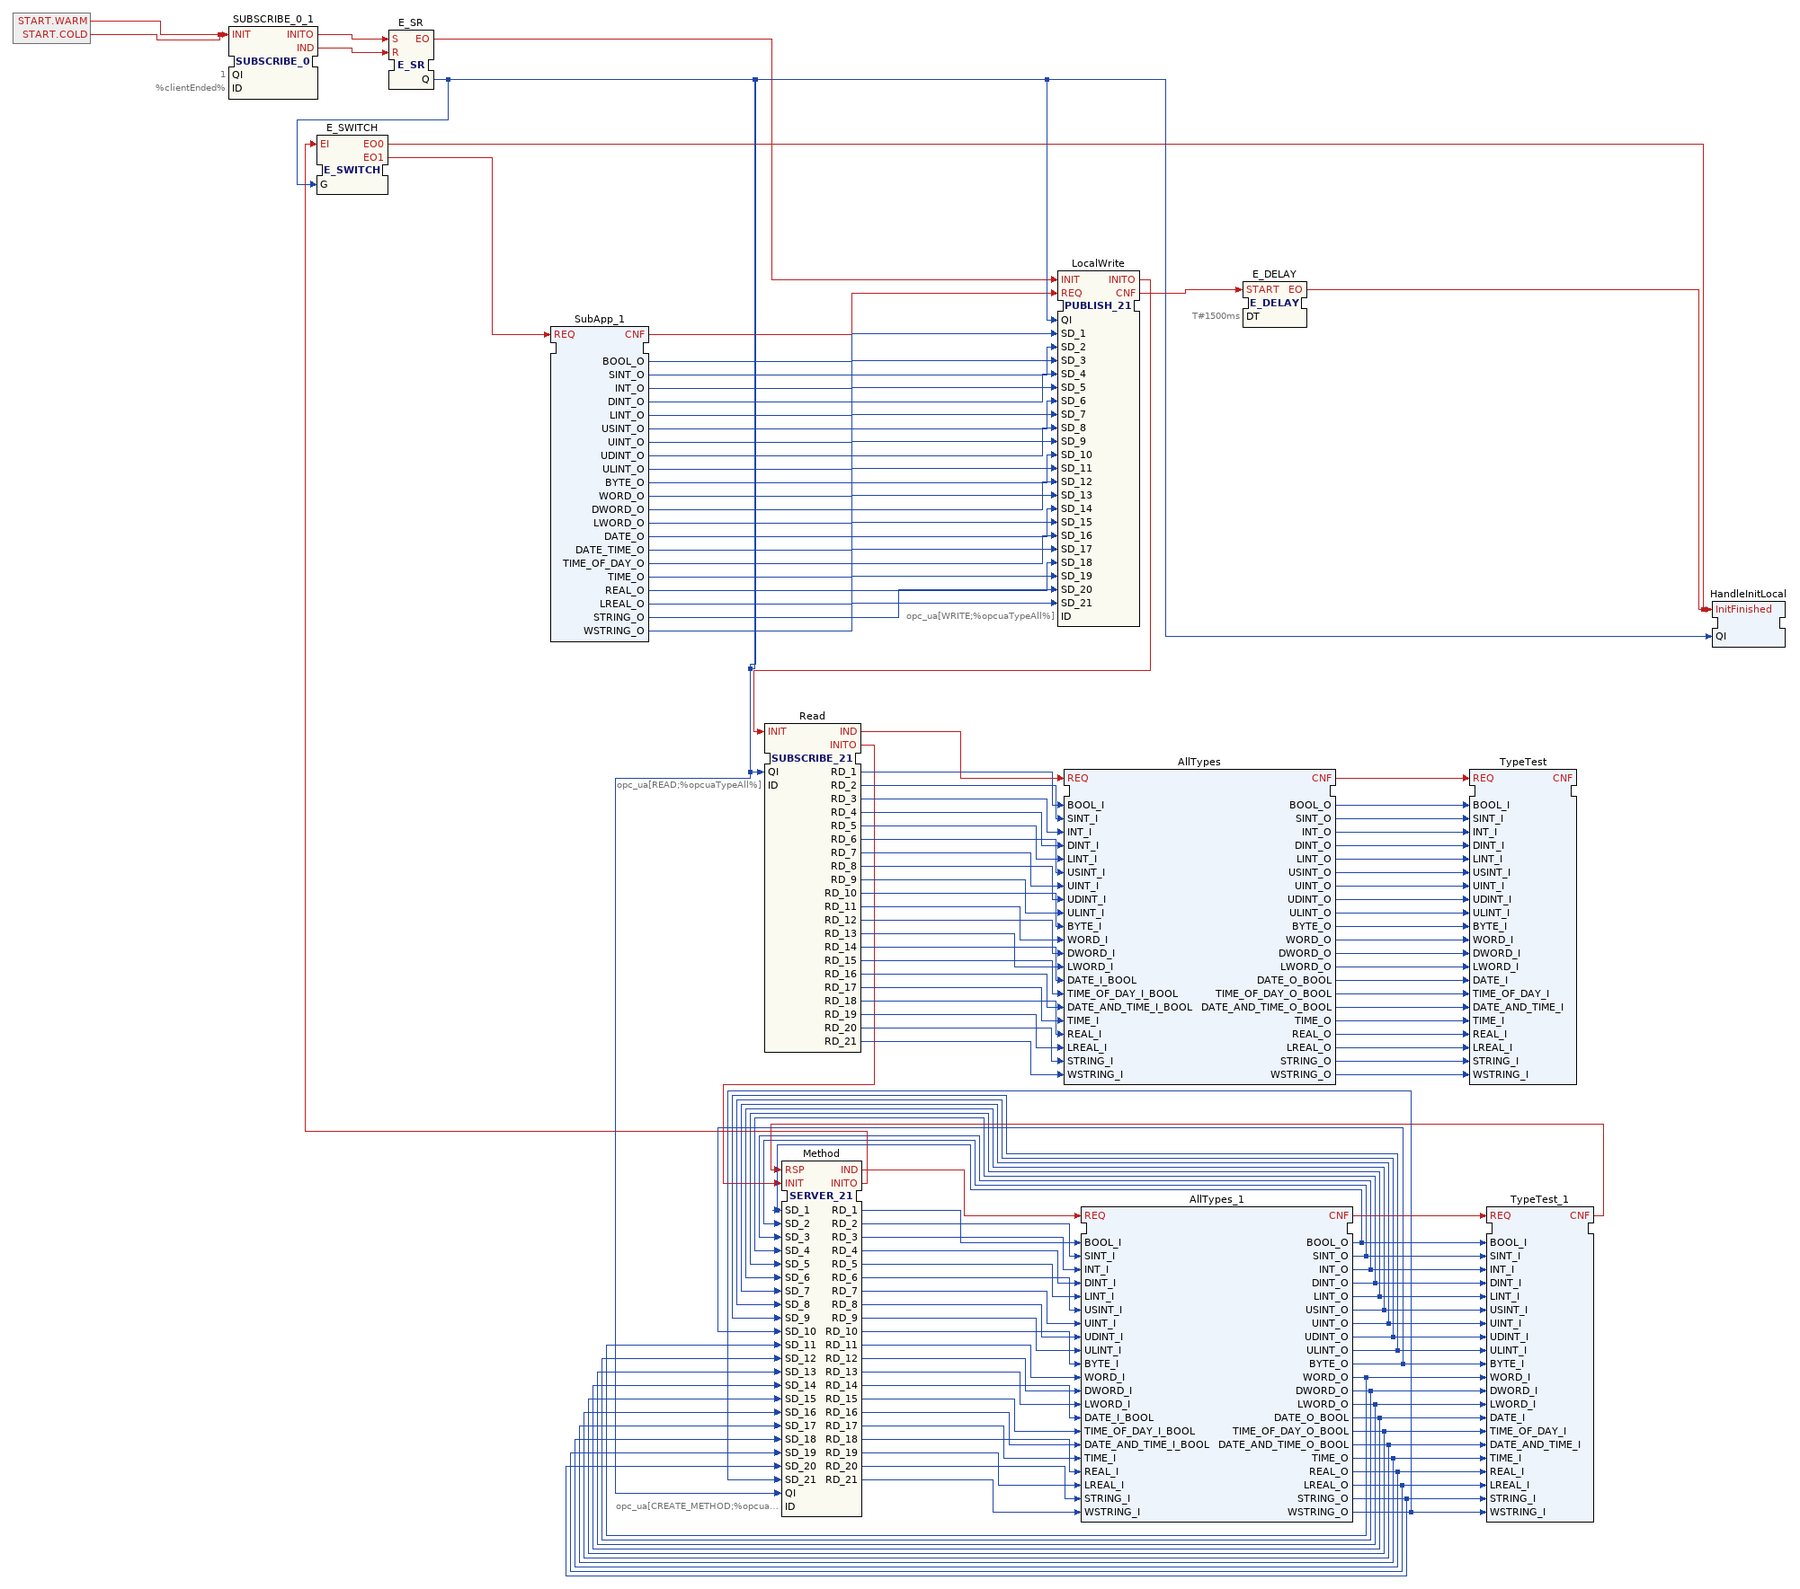
      FBS
        LocalWrite : PUBLISH_21(ID := opc_ua[WRITE;%opcuaTypeAll%]);
        Method : SERVER_21(ID := opc_ua[CREATE_METHOD;%opcuaTypeNode%]);
        Read : SUBSCRIBE_21(ID := opc_ua[READ;%opcuaTypeAll%]);
        E_SR : E_SR;
        SUBSCRIBE_0_1 : SUBSCRIBE_0(QI := 1, ID := %clientEnded%);
        E_SWITCH : E_SWITCH;
        E_DELAY : E_DELAY(DT := T#1500ms);
      END_FBS
      SUBAPPLICATION AllTypes
        EVENT_INPUT
          REQ;
        END_EVENT
        EVENT_OUTPUT
          CNF;
        END_EVENT
        VAR_INPUT
          BOOL_I : BOOL; (* BOOL Type Input *)
          SINT_I : SINT; (* SINT Type Input *)
          INT_I : INT; (* INT Type Input *)
          DINT_I : DINT; (* DINT Type Input *)
          LINT_I : LINT; (* LINT Type Input *)
          USINT_I : USINT; (* USINT Type Input *)
          UINT_I : UINT; (* UINT Type Input *)
          UDINT_I : UDINT; (* UDINT Type Input *)
          ULINT_I : ULINT; (* ULINT Type Input *)
          BYTE_I : BYTE; (* BYTE Type Input *)
          WORD_I : WORD; (* WORD Type Input *)
          DWORD_I : DWORD; (* DWORD Type Input *)
          LWORD_I : LWORD; (* LWORD Type Input *)
          DATE_I_BOOL : BOOL; (* DATE Type Input *)
          TIME_OF_DAY_I_BOOL : BOOL; (* TIME_OF_DAY Type Input *)
          DATE_AND_TIME_I_BOOL : BOOL; (* DATE_AND_TIME Type Input *)
          TIME_I : TIME; (* TIME Type Input *)
          REAL_I : REAL; (* REAL Type Input *)
          LREAL_I : LREAL; (* LREAL Type Input *)
          STRING_I : STRING; (* STRING Type Input *)
          WSTRING_I : WSTRING; (* WSTRING Type Input *)
        END_VAR
        VAR_OUTPUT
          BOOL_O : BOOL; (* BOOL Type Output *)
          SINT_O : SINT; (* SINT Type Output *)
          INT_O : INT; (* INT Type Output *)
          DINT_O : DINT; (* DINT Type Output *)
          LINT_O : LINT; (* LINT Type Output *)
          USINT_O : USINT; (* USINT Type Output *)
          UINT_O : UINT; (* UINT Type Output *)
          UDINT_O : UDINT; (* UDINT Type Output *)
          ULINT_O : ULINT; (* ULINT Type Output *)
          BYTE_O : BYTE; (* BYTE Type Output *)
          WORD_O : WORD; (* WORD Type Output *)
          DWORD_O : DWORD; (* DWORD Type Output *)
          LWORD_O : LWORD; (* LWORD Type Output *)
          DATE_O_BOOL : BOOL; (* DATE Type Output *)
          TIME_OF_DAY_O_BOOL : BOOL; (* TIME_OF_DAY Type Output *)
          DATE_AND_TIME_O_BOOL : BOOL; (* DATE_AND_TIME Type Output *)
          TIME_O : TIME; (* TIME Type Output *)
          REAL_O : REAL; (* REAL Type Output *)
          LREAL_O : LREAL; (* LREAL Type Output *)
          STRING_O : STRING; (* STRING Type Output *)
          WSTRING_O : WSTRING; (* WSTRING Type Output *)
        END_VAR
      END_SUBAPPLICATION
      SUBAPPLICATION TypeTest
        EVENT_INPUT
          REQ;
        END_EVENT
        EVENT_OUTPUT
          CNF;
        END_EVENT
        VAR_INPUT
          BOOL_I : BOOL; (* BOOL Type Input *)
          SINT_I : SINT; (* SINT Type Input *)
          INT_I : INT; (* INT Type Input *)
          DINT_I : DINT; (* DINT Type Input *)
          LINT_I : LINT; (* LINT Type Input *)
          USINT_I : USINT; (* USINT Type Input *)
          UINT_I : UINT; (* UINT Type Input *)
          UDINT_I : UDINT; (* UDINT Type Input *)
          ULINT_I : ULINT; (* ULINT Type Input *)
          BYTE_I : BYTE; (* BYTE Type Input *)
          WORD_I : WORD; (* WORD Type Input *)
          DWORD_I : DWORD; (* DWORD Type Input *)
          LWORD_I : LWORD; (* LWORD Type Input *)
          DATE_I : DATE; (* DATE Type Input *)
          TIME_OF_DAY_I : TIME_OF_DAY; (* TIME_OF_DAY Type Input *)
          DATE_AND_TIME_I : DATE_AND_TIME; (* DATE_AND_TIME Type Input *)
          TIME_I : TIME; (* TIME Type Input *)
          REAL_I : REAL; (* REAL Type Input *)
          LREAL_I : LREAL; (* LREAL Type Input *)
          STRING_I : STRING; (* STRING Type Input *)
          WSTRING_I : WSTRING; (* WSTRING Type Input *)
        END_VAR
      END_SUBAPPLICATION
      SUBAPPLICATION AllTypes_1
        EVENT_INPUT
          REQ;
        END_EVENT
        EVENT_OUTPUT
          CNF;
        END_EVENT
        VAR_INPUT
          BOOL_I : BOOL; (* BOOL Type Input *)
          SINT_I : SINT; (* SINT Type Input *)
          INT_I : INT; (* INT Type Input *)
          DINT_I : DINT; (* DINT Type Input *)
          LINT_I : LINT; (* LINT Type Input *)
          USINT_I : USINT; (* USINT Type Input *)
          UINT_I : UINT; (* UINT Type Input *)
          UDINT_I : UDINT; (* UDINT Type Input *)
          ULINT_I : ULINT; (* ULINT Type Input *)
          BYTE_I : BYTE; (* BYTE Type Input *)
          WORD_I : WORD; (* WORD Type Input *)
          DWORD_I : DWORD; (* DWORD Type Input *)
          LWORD_I : LWORD; (* LWORD Type Input *)
          DATE_I_BOOL : BOOL; (* DATE Type Input *)
          TIME_OF_DAY_I_BOOL : BOOL; (* TIME_OF_DAY Type Input *)
          DATE_AND_TIME_I_BOOL : BOOL; (* DATE_AND_TIME Type Input *)
          TIME_I : TIME; (* TIME Type Input *)
          REAL_I : REAL; (* REAL Type Input *)
          LREAL_I : LREAL; (* LREAL Type Input *)
          STRING_I : STRING; (* STRING Type Input *)
          WSTRING_I : WSTRING; (* WSTRING Type Input *)
        END_VAR
        VAR_OUTPUT
          BOOL_O : BOOL; (* BOOL Type Output *)
          SINT_O : SINT; (* SINT Type Output *)
          INT_O : INT; (* INT Type Output *)
          DINT_O : DINT; (* DINT Type Output *)
          LINT_O : LINT; (* LINT Type Output *)
          USINT_O : USINT; (* USINT Type Output *)
          UINT_O : UINT; (* UINT Type Output *)
          UDINT_O : UDINT; (* UDINT Type Output *)
          ULINT_O : ULINT; (* ULINT Type Output *)
          BYTE_O : BYTE; (* BYTE Type Output *)
          WORD_O : WORD; (* WORD Type Output *)
          DWORD_O : DWORD; (* DWORD Type Output *)
          LWORD_O : LWORD; (* LWORD Type Output *)
          DATE_O_BOOL : BOOL; (* DATE Type Output *)
          TIME_OF_DAY_O_BOOL : BOOL; (* TIME_OF_DAY Type Output *)
          DATE_AND_TIME_O_BOOL : BOOL; (* DATE_AND_TIME Type Output *)
          TIME_O : TIME; (* TIME Type Output *)
          REAL_O : REAL; (* REAL Type Output *)
          LREAL_O : LREAL; (* LREAL Type Output *)
          STRING_O : STRING; (* STRING Type Output *)
          WSTRING_O : WSTRING; (* WSTRING Type Output *)
        END_VAR
      END_SUBAPPLICATION
      SUBAPPLICATION TypeTest_1
        EVENT_INPUT
          REQ;
        END_EVENT
        EVENT_OUTPUT
          CNF;
        END_EVENT
        VAR_INPUT
          BOOL_I : BOOL; (* BOOL Type Input *)
          SINT_I : SINT; (* SINT Type Input *)
          INT_I : INT; (* INT Type Input *)
          DINT_I : DINT; (* DINT Type Input *)
          LINT_I : LINT; (* LINT Type Input *)
          USINT_I : USINT; (* USINT Type Input *)
          UINT_I : UINT; (* UINT Type Input *)
          UDINT_I : UDINT; (* UDINT Type Input *)
          ULINT_I : ULINT; (* ULINT Type Input *)
          BYTE_I : BYTE; (* BYTE Type Input *)
          WORD_I : WORD; (* WORD Type Input *)
          DWORD_I : DWORD; (* DWORD Type Input *)
          LWORD_I : LWORD; (* LWORD Type Input *)
          DATE_I : DATE; (* DATE Type Input *)
          TIME_OF_DAY_I : TIME_OF_DAY; (* TIME_OF_DAY Type Input *)
          DATE_AND_TIME_I : DATE_AND_TIME; (* DATE_AND_TIME Type Input *)
          TIME_I : TIME; (* TIME Type Input *)
          REAL_I : REAL; (* REAL Type Input *)
          LREAL_I : LREAL; (* LREAL Type Input *)
          STRING_I : STRING; (* STRING Type Input *)
          WSTRING_I : WSTRING; (* WSTRING Type Input *)
        END_VAR
      END_SUBAPPLICATION
      SUBAPPLICATION HandleInitLocal
        EVENT_INPUT
          InitFinished;
        END_EVENT
        VAR_INPUT
          QI : BOOL;
        END_VAR
      END_SUBAPPLICATION
      SUBAPPLICATION SubApp_1
        EVENT_INPUT
          REQ;
        END_EVENT
        EVENT_OUTPUT
          CNF;
        END_EVENT
        VAR_OUTPUT
          BOOL_O : BOOL;
          SINT_O : SINT;
          INT_O : INT;
          DINT_O : DINT;
          LINT_O : LINT;
          USINT_O : USINT;
          UINT_O : UINT;
          UDINT_O : UDINT;
          ULINT_O : ULINT;
          BYTE_O : BYTE;
          WORD_O : WORD;
          DWORD_O : DWORD;
          LWORD_O : LWORD;
          DATE_O : BOOL;
          DATE_TIME_O : BOOL;
          TIME_OF_DAY_O : BOOL;
          TIME_O : TIME;
          REAL_O : REAL;
          LREAL_O : LREAL;
          STRING_O : STRING;
          WSTRING_O : WSTRING;
        END_VAR
      END_SUBAPPLICATION
      EVENT_CONNECTIONS
        AllTypes.CNF TO TypeTest.REQ;
        Method.IND TO AllTypes_1.REQ;
        Read.IND TO AllTypes.REQ;
        AllTypes_1.CNF TO TypeTest_1.REQ;
        TypeTest_1.CNF TO Method.RSP;
        SUBSCRIBE_0_1.INITO TO E_SR.S;
        SUBSCRIBE_0_1.IND TO E_SR.R;
        LocalWrite.INITO TO Read.INIT;
        Read.INITO TO Method.INIT;
        START.WARM TO SUBSCRIBE_0_1.INIT;
        START.COLD TO SUBSCRIBE_0_1.INIT;
        E_SR.EO TO LocalWrite.INIT;
        Method.INITO TO E_SWITCH.EI;
        E_SWITCH.EO0 TO HandleInitLocal.InitFinished;
        LocalWrite.CNF TO E_DELAY.START;
        E_DELAY.EO TO HandleInitLocal.InitFinished;
        SubApp_1.CNF TO LocalWrite.REQ;
        E_SWITCH.EO1 TO SubApp_1.REQ;
      END_CONNECTIONS
      DATA_CONNECTIONS
        AllTypes.BOOL_O TO TypeTest.BOOL_I;
        AllTypes.SINT_O TO TypeTest.SINT_I;
        AllTypes.INT_O TO TypeTest.INT_I;
        AllTypes.DINT_O TO TypeTest.DINT_I;
        AllTypes.LINT_O TO TypeTest.LINT_I;
        AllTypes.USINT_O TO TypeTest.USINT_I;
        AllTypes.UINT_O TO TypeTest.UINT_I;
        AllTypes.UDINT_O TO TypeTest.UDINT_I;
        AllTypes.ULINT_O TO TypeTest.ULINT_I;
        AllTypes.BYTE_O TO TypeTest.BYTE_I;
        AllTypes.WORD_O TO TypeTest.WORD_I;
        AllTypes.DWORD_O TO TypeTest.DWORD_I;
        AllTypes.LWORD_O TO TypeTest.LWORD_I;
        AllTypes.DATE_O_BOOL TO TypeTest.DATE_I;
        AllTypes.TIME_OF_DAY_O_BOOL TO TypeTest.TIME_OF_DAY_I;
        AllTypes.DATE_AND_TIME_O_BOOL TO TypeTest.DATE_AND_TIME_I;
        AllTypes.TIME_O TO TypeTest.TIME_I;
        AllTypes.REAL_O TO TypeTest.REAL_I;
        AllTypes.LREAL_O TO TypeTest.LREAL_I;
        AllTypes.STRING_O TO TypeTest.STRING_I;
        AllTypes.WSTRING_O TO TypeTest.WSTRING_I;
        Method.RD_1 TO AllTypes_1.BOOL_I;
        Method.RD_2 TO AllTypes_1.SINT_I;
        Method.RD_3 TO AllTypes_1.INT_I;
        Method.RD_4 TO AllTypes_1.DINT_I;
        Method.RD_5 TO AllTypes_1.LINT_I;
        Method.RD_6 TO AllTypes_1.USINT_I;
        Method.RD_7 TO AllTypes_1.UINT_I;
        Method.RD_8 TO AllTypes_1.UDINT_I;
        Method.RD_9 TO AllTypes_1.ULINT_I;
        Method.RD_10 TO AllTypes_1.BYTE_I;
        Method.RD_11 TO AllTypes_1.WORD_I;
        Method.RD_12 TO AllTypes_1.DWORD_I;
        Method.RD_13 TO AllTypes_1.LWORD_I;
        Method.RD_14 TO AllTypes_1.DATE_I_BOOL;
        Method.RD_15 TO AllTypes_1.TIME_OF_DAY_I_BOOL;
        Method.RD_16 TO AllTypes_1.DATE_AND_TIME_I_BOOL;
        Method.RD_17 TO AllTypes_1.TIME_I;
        Method.RD_18 TO AllTypes_1.REAL_I;
        Method.RD_19 TO AllTypes_1.LREAL_I;
        Method.RD_20 TO AllTypes_1.STRING_I;
        Method.RD_21 TO AllTypes_1.WSTRING_I;
        AllTypes_1.BOOL_O TO Method.SD_1;
        AllTypes_1.SINT_O TO Method.SD_2;
        AllTypes_1.INT_O TO Method.SD_3;
        AllTypes_1.DINT_O TO Method.SD_4;
        AllTypes_1.LINT_O TO Method.SD_5;
        AllTypes_1.USINT_O TO Method.SD_6;
        AllTypes_1.UINT_O TO Method.SD_7;
        AllTypes_1.UDINT_O TO Method.SD_8;
        AllTypes_1.ULINT_O TO Method.SD_9;
        AllTypes_1.BYTE_O TO Method.SD_10;
        AllTypes_1.WORD_O TO Method.SD_11;
        AllTypes_1.DWORD_O TO Method.SD_12;
        AllTypes_1.LWORD_O TO Method.SD_13;
        AllTypes_1.DATE_O_BOOL TO Method.SD_14;
        AllTypes_1.TIME_OF_DAY_O_BOOL TO Method.SD_15;
        AllTypes_1.DATE_AND_TIME_O_BOOL TO Method.SD_16;
        AllTypes_1.TIME_O TO Method.SD_17;
        AllTypes_1.REAL_O TO Method.SD_18;
        AllTypes_1.LREAL_O TO Method.SD_19;
        AllTypes_1.STRING_O TO Method.SD_20;
        AllTypes_1.WSTRING_O TO Method.SD_21;
        Read.RD_1 TO AllTypes.BOOL_I;
        Read.RD_2 TO AllTypes.SINT_I;
        Read.RD_3 TO AllTypes.INT_I;
        Read.RD_4 TO AllTypes.DINT_I;
        Read.RD_5 TO AllTypes.LINT_I;
        Read.RD_6 TO AllTypes.USINT_I;
        Read.RD_7 TO AllTypes.UINT_I;
        Read.RD_8 TO AllTypes.UDINT_I;
        Read.RD_9 TO AllTypes.ULINT_I;
        Read.RD_10 TO AllTypes.BYTE_I;
        Read.RD_11 TO AllTypes.WORD_I;
        Read.RD_12 TO AllTypes.DWORD_I;
        Read.RD_13 TO AllTypes.LWORD_I;
        Read.RD_14 TO AllTypes.DATE_I_BOOL;
        Read.RD_15 TO AllTypes.TIME_OF_DAY_I_BOOL;
        Read.RD_16 TO AllTypes.DATE_AND_TIME_I_BOOL;
        Read.RD_17 TO AllTypes.TIME_I;
        Read.RD_18 TO AllTypes.REAL_I;
        Read.RD_19 TO AllTypes.LREAL_I;
        Read.RD_20 TO AllTypes.STRING_I;
        Read.RD_21 TO AllTypes.WSTRING_I;
        AllTypes_1.BOOL_O TO TypeTest_1.BOOL_I;
        AllTypes_1.SINT_O TO TypeTest_1.SINT_I;
        AllTypes_1.INT_O TO TypeTest_1.INT_I;
        AllTypes_1.DINT_O TO TypeTest_1.DINT_I;
        AllTypes_1.LINT_O TO TypeTest_1.LINT_I;
        AllTypes_1.USINT_O TO TypeTest_1.USINT_I;
        AllTypes_1.UINT_O TO TypeTest_1.UINT_I;
        AllTypes_1.UDINT_O TO TypeTest_1.UDINT_I;
        AllTypes_1.ULINT_O TO TypeTest_1.ULINT_I;
        AllTypes_1.BYTE_O TO TypeTest_1.BYTE_I;
        AllTypes_1.WORD_O TO TypeTest_1.WORD_I;
        AllTypes_1.DWORD_O TO TypeTest_1.DWORD_I;
        AllTypes_1.LWORD_O TO TypeTest_1.LWORD_I;
        AllTypes_1.DATE_O_BOOL TO TypeTest_1.DATE_I;
        AllTypes_1.TIME_OF_DAY_O_BOOL TO TypeTest_1.TIME_OF_DAY_I;
        AllTypes_1.DATE_AND_TIME_O_BOOL TO TypeTest_1.DATE_AND_TIME_I;
        AllTypes_1.TIME_O TO TypeTest_1.TIME_I;
        AllTypes_1.REAL_O TO TypeTest_1.REAL_I;
        AllTypes_1.LREAL_O TO TypeTest_1.LREAL_I;
        AllTypes_1.STRING_O TO TypeTest_1.STRING_I;
        AllTypes_1.WSTRING_O TO TypeTest_1.WSTRING_I;
        E_SR.Q TO HandleInitLocal.QI;
        E_SR.Q TO LocalWrite.QI;
        E_SR.Q TO Read.QI;
        E_SR.Q TO Method.QI;
        E_SR.Q TO E_SWITCH.G;
        SubApp_1.BOOL_O TO LocalWrite.SD_1;
        SubApp_1.SINT_O TO LocalWrite.SD_2;
        SubApp_1.INT_O TO LocalWrite.SD_3;
        SubApp_1.DINT_O TO LocalWrite.SD_4;
        SubApp_1.LINT_O TO LocalWrite.SD_5;
        SubApp_1.USINT_O TO LocalWrite.SD_6;
        SubApp_1.UINT_O TO LocalWrite.SD_7;
        SubApp_1.UDINT_O TO LocalWrite.SD_8;
        SubApp_1.ULINT_O TO LocalWrite.SD_9;
        SubApp_1.BYTE_O TO LocalWrite.SD_10;
        SubApp_1.WORD_O TO LocalWrite.SD_11;
        SubApp_1.DWORD_O TO LocalWrite.SD_12;
        SubApp_1.LWORD_O TO LocalWrite.SD_13;
        SubApp_1.DATE_O TO LocalWrite.SD_14;
        SubApp_1.DATE_TIME_O TO LocalWrite.SD_15;
        SubApp_1.TIME_OF_DAY_O TO LocalWrite.SD_16;
        SubApp_1.TIME_O TO LocalWrite.SD_17;
        SubApp_1.REAL_O TO LocalWrite.SD_18;
        SubApp_1.LREAL_O TO LocalWrite.SD_19;
        SubApp_1.STRING_O TO LocalWrite.SD_20;
        SubApp_1.WSTRING_O TO LocalWrite.SD_21;
      END_CONNECTIONS
    END_RESOURCE
    RESOURCE TestServer : EMB_RES
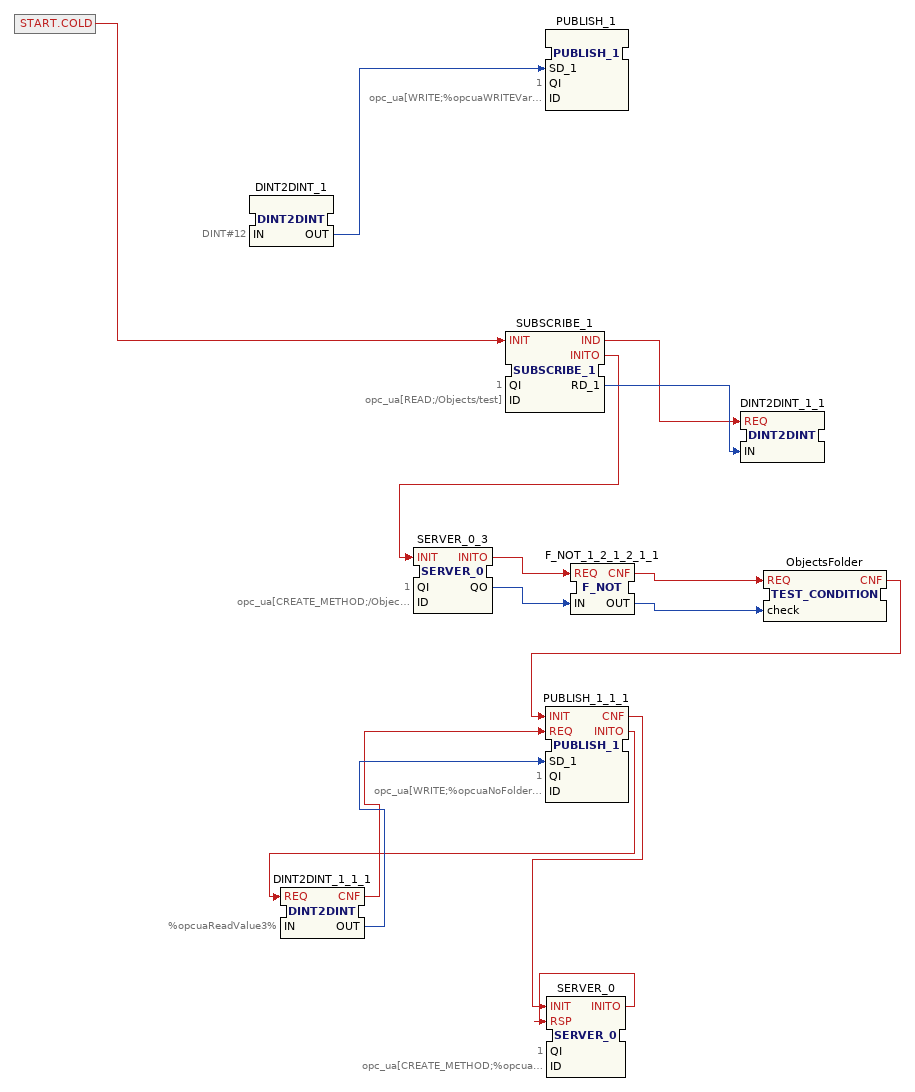
      FBS
        DINT2DINT_1 : DINT2DINT(IN := DINT#12);
        PUBLISH_1 : PUBLISH_1(QI := 1, ID := opc_ua[WRITE;%opcuaWRITEVariable%]);
        SUBSCRIBE_1 : SUBSCRIBE_1(QI := 1, ID := opc_ua[READ;/Objects/test]);
        DINT2DINT_1_1 : DINT2DINT;
        F_NOT_1_2_1_2_1_1 : F_NOT;
        ObjectsFolder : TEST_CONDITION;
        SERVER_0_3 : SERVER_0(QI := 1, ID := opc_ua[CREATE_METHOD;/Objects]);
        PUBLISH_1_1_1 : PUBLISH_1(QI := 1, ID := opc_ua[WRITE;%opcuaNoFolder%]);
        SERVER_0 : SERVER_0(QI := 1, ID := opc_ua[CREATE_METHOD;%opcuaNoFolderMethod%]);
        DINT2DINT_1_1_1 : DINT2DINT(IN := %opcuaReadValue3%);
      END_FBS
      EVENT_CONNECTIONS
        SUBSCRIBE_1.IND TO DINT2DINT_1_1.REQ;
        START.COLD TO SUBSCRIBE_1.INIT;
        F_NOT_1_2_1_2_1_1.CNF TO ObjectsFolder.REQ;
        SERVER_0_3.INITO TO F_NOT_1_2_1_2_1_1.REQ;
        SUBSCRIBE_1.INITO TO SERVER_0_3.INIT;
        ObjectsFolder.CNF TO PUBLISH_1_1_1.INIT;
        PUBLISH_1_1_1.CNF TO SERVER_0.INIT;
        DINT2DINT_1_1_1.CNF TO PUBLISH_1_1_1.REQ;
        SERVER_0.INITO TO SERVER_0.RSP;
        PUBLISH_1_1_1.INITO TO DINT2DINT_1_1_1.REQ;
      END_CONNECTIONS
      DATA_CONNECTIONS
        DINT2DINT_1.OUT TO PUBLISH_1.SD_1;
        SUBSCRIBE_1.RD_1 TO DINT2DINT_1_1.IN;
        F_NOT_1_2_1_2_1_1.OUT TO ObjectsFolder.check;
        SERVER_0_3.QO TO F_NOT_1_2_1_2_1_1.IN;
        DINT2DINT_1_1_1.OUT TO PUBLISH_1_1_1.SD_1;
      END_CONNECTIONS
    END_RESOURCE
  END_DEVICE
  DEVICE OPCUACLient : FORTE_PC(MGR_ID := "localhost:61499")
    {SET_ATTRIBUTE(Profile, HOLOBLOC)} (* device profile *)
    RESOURCE WorkingClient : EMB_RES
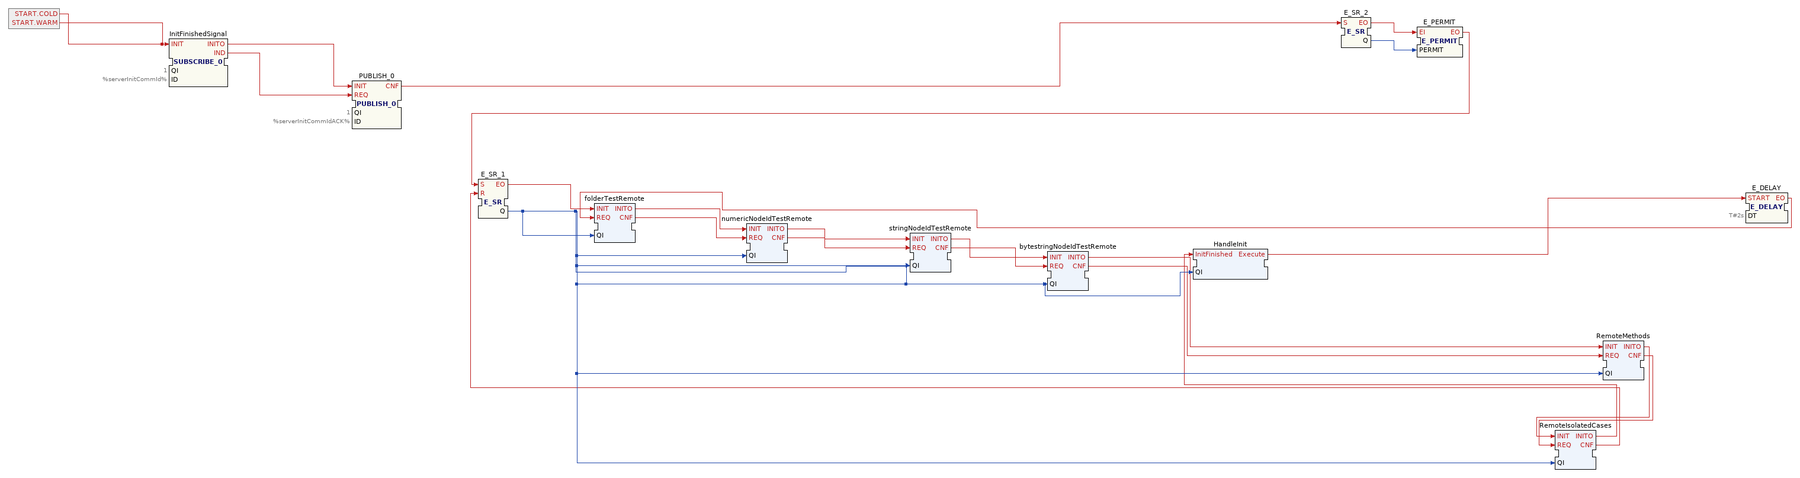
      FBS
        E_SR_1 : E_SR;
        InitFinishedSignal : SUBSCRIBE_0(QI := 1, ID := %serverInitCommId%);
        PUBLISH_0 : PUBLISH_0(QI := 1, ID := %serverInitCommIdACK%);
        E_SR_2 : E_SR;
        E_PERMIT : E_PERMIT;
        E_DELAY : E_DELAY(DT := T#2s);
      END_FBS
      SUBAPPLICATION folderTestRemote
        EVENT_INPUT
          INIT;
          REQ;
        END_EVENT
        EVENT_OUTPUT
          INITO;
          CNF;
        END_EVENT
        VAR_INPUT
          QI : BOOL;
        END_VAR
      END_SUBAPPLICATION
      SUBAPPLICATION HandleInit
        EVENT_INPUT
          InitFinished;
        END_EVENT
        EVENT_OUTPUT
          Execute;
        END_EVENT
        VAR_INPUT
          QI : BOOL;
        END_VAR
      END_SUBAPPLICATION
      SUBAPPLICATION numericNodeIdTestRemote
        EVENT_INPUT
          INIT;
          REQ;
        END_EVENT
        EVENT_OUTPUT
          INITO;
          CNF;
        END_EVENT
        VAR_INPUT
          QI : BOOL;
        END_VAR
      END_SUBAPPLICATION
      SUBAPPLICATION stringNodeIdTestRemote
        EVENT_INPUT
          INIT;
          REQ;
        END_EVENT
        EVENT_OUTPUT
          INITO;
          CNF;
        END_EVENT
        VAR_INPUT
          QI : BOOL;
        END_VAR
      END_SUBAPPLICATION
      SUBAPPLICATION bytestringNodeIdTestRemote
        EVENT_INPUT
          INIT;
          REQ;
        END_EVENT
        EVENT_OUTPUT
          INITO;
          CNF;
        END_EVENT
        VAR_INPUT
          QI : BOOL;
        END_VAR
      END_SUBAPPLICATION
      SUBAPPLICATION RemoteMethods
        EVENT_INPUT
          INIT;
          REQ;
        END_EVENT
        EVENT_OUTPUT
          INITO;
          CNF;
        END_EVENT
        VAR_INPUT
          QI : BOOL;
        END_VAR
      END_SUBAPPLICATION
      SUBAPPLICATION RemoteIsolatedCases
        EVENT_INPUT
          INIT;
          REQ;
        END_EVENT
        EVENT_OUTPUT
          INITO;
          CNF;
        END_EVENT
        VAR_INPUT
          QI : BOOL;
        END_VAR
      END_SUBAPPLICATION
      EVENT_CONNECTIONS
        START.COLD TO InitFinishedSignal.INIT;
        START.WARM TO InitFinishedSignal.INIT;
        InitFinishedSignal.INITO TO PUBLISH_0.INIT;
        folderTestRemote.INITO TO numericNodeIdTestRemote.INIT;
        numericNodeIdTestRemote.INITO TO stringNodeIdTestRemote.INIT;
        stringNodeIdTestRemote.INITO TO bytestringNodeIdTestRemote.INIT;
        InitFinishedSignal.IND TO PUBLISH_0.REQ;
        PUBLISH_0.CNF TO E_SR_2.S;
        E_SR_2.EO TO E_PERMIT.EI;
        E_PERMIT.EO TO E_SR_1.S;
        E_DELAY.EO TO folderTestRemote.REQ;
        HandleInit.Execute TO E_DELAY.START;
        bytestringNodeIdTestRemote.INITO TO RemoteMethods.INIT;
        E_SR_1.EO TO folderTestRemote.INIT;
        bytestringNodeIdTestRemote.CNF TO RemoteMethods.REQ;
        stringNodeIdTestRemote.CNF TO bytestringNodeIdTestRemote.REQ;
        numericNodeIdTestRemote.CNF TO stringNodeIdTestRemote.REQ;
        folderTestRemote.CNF TO numericNodeIdTestRemote.REQ;
        RemoteIsolatedCases.INITO TO HandleInit.InitFinished;
        RemoteMethods.INITO TO RemoteIsolatedCases.INIT;
        RemoteIsolatedCases.CNF TO E_SR_1.R;
        RemoteMethods.CNF TO RemoteIsolatedCases.REQ;
      END_CONNECTIONS
      DATA_CONNECTIONS
        E_SR_1.Q TO folderTestRemote.QI;
        E_SR_1.Q TO HandleInit.QI;
        E_SR_1.Q TO numericNodeIdTestRemote.QI;
        E_SR_1.Q TO stringNodeIdTestRemote.QI;
        E_SR_1.Q TO bytestringNodeIdTestRemote.QI;
        E_SR_2.Q TO E_PERMIT.PERMIT;
        E_SR_1.Q TO RemoteMethods.QI;
        E_SR_1.Q TO RemoteIsolatedCases.QI;
      END_CONNECTIONS
    END_RESOURCE
    RESOURCE WokingClientWithoutSubs : EMB_RES
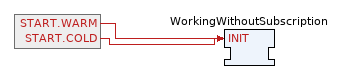
      SUBAPPLICATION WorkingWithoutSubscription
        EVENT_INPUT
          INIT;
        END_EVENT
      END_SUBAPPLICATION
      EVENT_CONNECTIONS
        START.WARM TO WorkingWithoutSubscription.INIT;
        START.COLD TO WorkingWithoutSubscription.INIT;
      END_CONNECTIONS
    END_RESOURCE
    RESOURCE FailingClient : EMB_RES
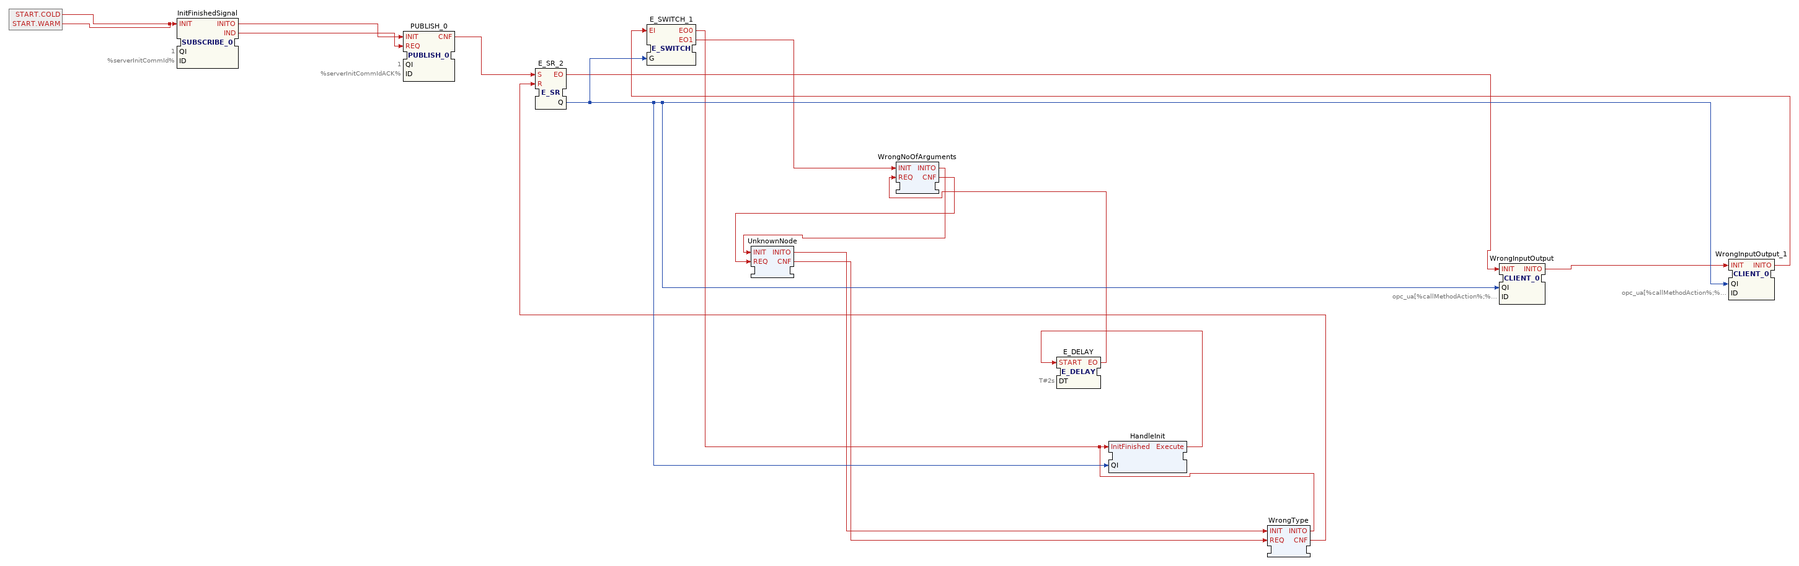
      FBS
        E_SWITCH_1 : E_SWITCH;
        InitFinishedSignal : SUBSCRIBE_0(QI := 1, ID := %serverInitCommId%);
        E_DELAY : E_DELAY(DT := T#2s);
        E_SR_2 : E_SR;
        PUBLISH_0 : PUBLISH_0(QI := 1, ID := %serverInitCommIdACK%);
        WrongInputOutput : CLIENT_0(ID := opc_ua[%callMethodAction%;%unknownEndpoint%;%opcuaMethodCreation7%]);
        WrongInputOutput_1 : CLIENT_0(ID := opc_ua[%callMethodAction%;%unknownEndpoint%;%opcuaMethodCreation7%]);
      END_FBS
      SUBAPPLICATION HandleInit
        EVENT_INPUT
          InitFinished;
        END_EVENT
        EVENT_OUTPUT
          Execute;
        END_EVENT
        VAR_INPUT
          QI : BOOL;
        END_VAR
      END_SUBAPPLICATION
      SUBAPPLICATION UnknownNode
        EVENT_INPUT
          INIT;
          REQ;
        END_EVENT
        EVENT_OUTPUT
          INITO;
          CNF;
        END_EVENT
      END_SUBAPPLICATION
      SUBAPPLICATION WrongNoOfArguments
        EVENT_INPUT
          INIT;
          REQ;
        END_EVENT
        EVENT_OUTPUT
          INITO;
          CNF;
        END_EVENT
      END_SUBAPPLICATION
      SUBAPPLICATION WrongType
        EVENT_INPUT
          INIT;
          REQ;
        END_EVENT
        EVENT_OUTPUT
          INITO;
          CNF;
        END_EVENT
      END_SUBAPPLICATION
      EVENT_CONNECTIONS
        E_SWITCH_1.EO0 TO HandleInit.InitFinished;
        HandleInit.Execute TO E_DELAY.START;
        InitFinishedSignal.INITO TO PUBLISH_0.INIT;
        InitFinishedSignal.IND TO PUBLISH_0.REQ;
        PUBLISH_0.CNF TO E_SR_2.S;
        START.COLD TO InitFinishedSignal.INIT;
        START.WARM TO InitFinishedSignal.INIT;
        E_DELAY.EO TO WrongNoOfArguments.REQ;
        WrongNoOfArguments.CNF TO UnknownNode.REQ;
        WrongNoOfArguments.INITO TO UnknownNode.INIT;
        UnknownNode.INITO TO WrongType.INIT;
        UnknownNode.CNF TO WrongType.REQ;
        WrongType.INITO TO HandleInit.InitFinished;
        WrongType.CNF TO E_SR_2.R;
        WrongInputOutput.INITO TO WrongInputOutput_1.INIT;
        E_SR_2.EO TO WrongInputOutput.INIT;
        E_SWITCH_1.EO1 TO WrongNoOfArguments.INIT;
        WrongInputOutput_1.INITO TO E_SWITCH_1.EI;
      END_CONNECTIONS
      DATA_CONNECTIONS
        E_SR_2.Q TO HandleInit.QI;
        E_SR_2.Q TO E_SWITCH_1.G;
        E_SR_2.Q TO WrongInputOutput.QI;
        E_SR_2.Q TO WrongInputOutput_1.QI;
      END_CONNECTIONS
    END_RESOURCE
    RESOURCE delayedWorkingClient : EMB_RES
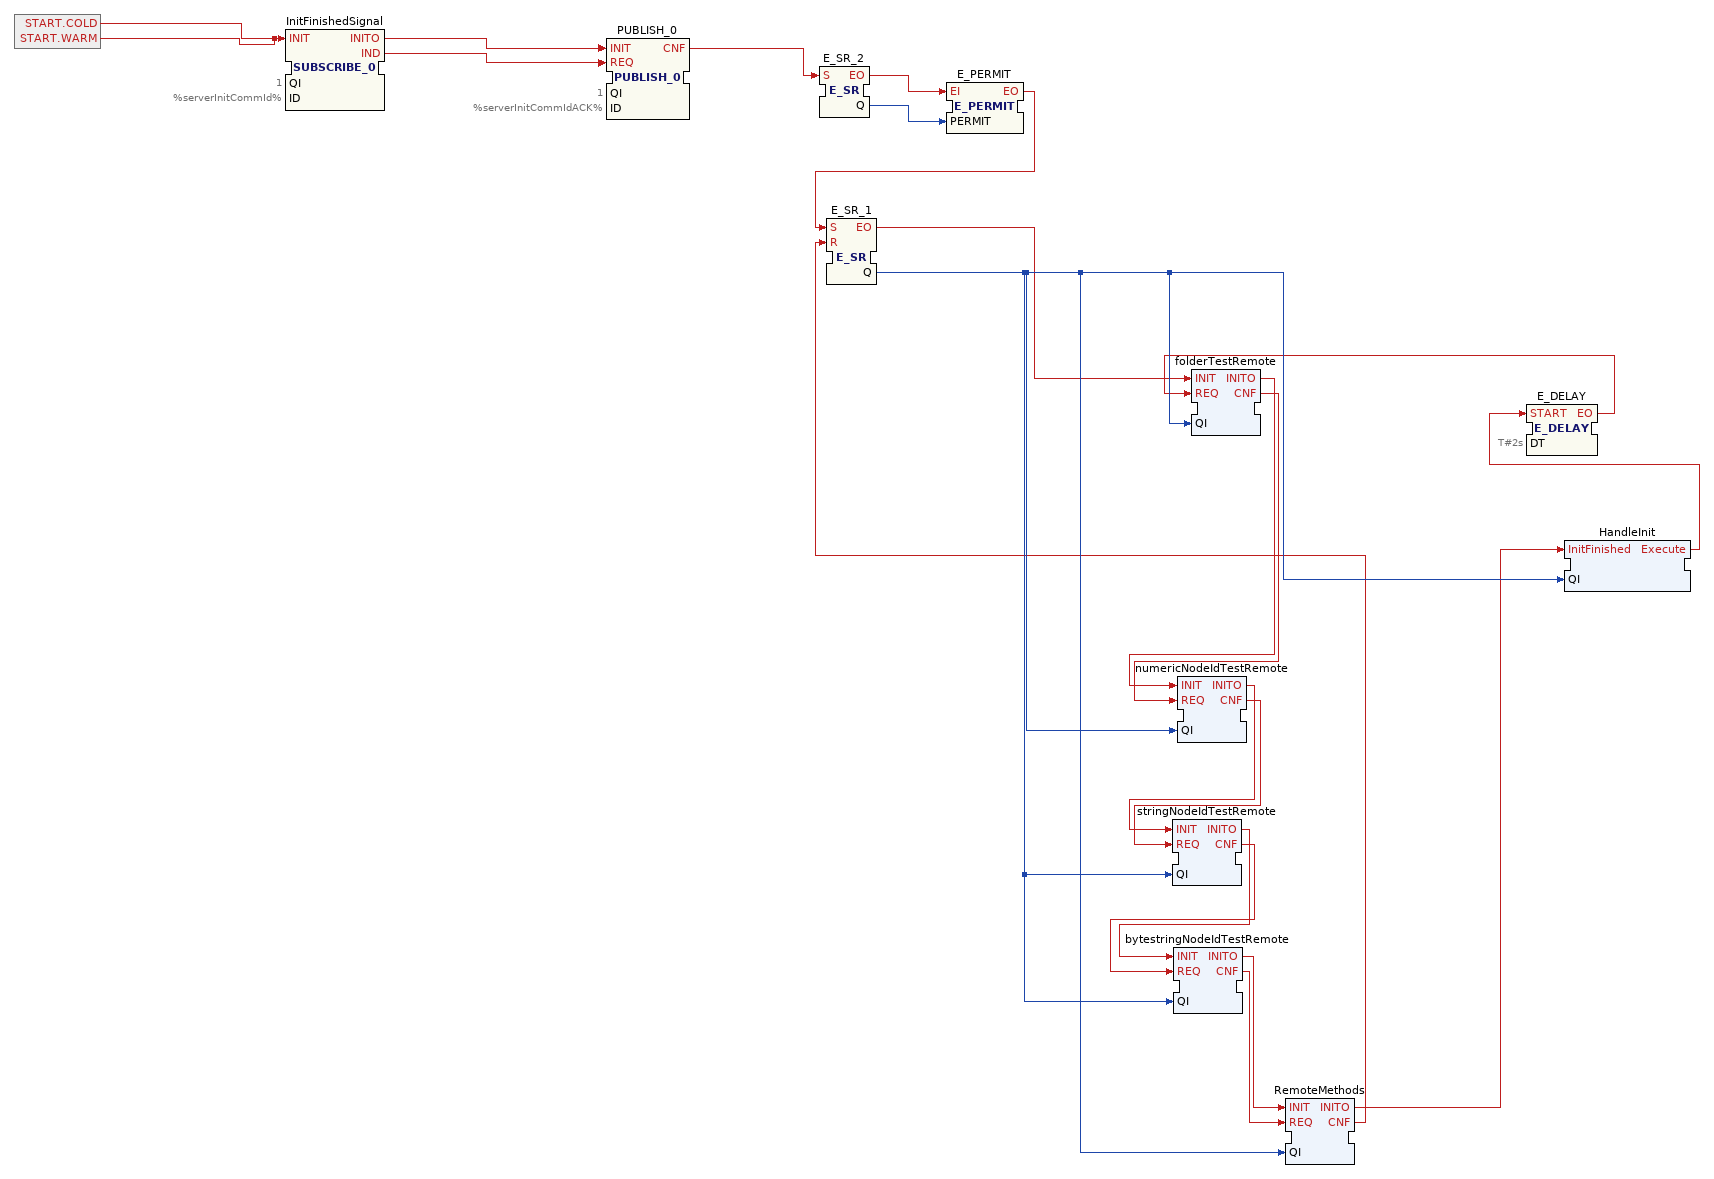
      FBS
        E_PERMIT : E_PERMIT;
        PUBLISH_0 : PUBLISH_0(QI := 1, ID := %serverInitCommIdACK%);
        InitFinishedSignal : SUBSCRIBE_0(QI := 1, ID := %serverInitCommId%);
        E_DELAY : E_DELAY(DT := T#2s);
        E_SR_1 : E_SR;
        E_SR_2 : E_SR;
      END_FBS
      SUBAPPLICATION numericNodeIdTestRemote
        EVENT_INPUT
          INIT;
          REQ;
        END_EVENT
        EVENT_OUTPUT
          INITO;
          CNF;
        END_EVENT
        VAR_INPUT
          QI : BOOL;
        END_VAR
      END_SUBAPPLICATION
      SUBAPPLICATION RemoteMethods
        EVENT_INPUT
          INIT;
          REQ;
        END_EVENT
        EVENT_OUTPUT
          INITO;
          CNF;
        END_EVENT
        VAR_INPUT
          QI : BOOL;
        END_VAR
      END_SUBAPPLICATION
      SUBAPPLICATION HandleInit
        EVENT_INPUT
          InitFinished;
        END_EVENT
        EVENT_OUTPUT
          Execute;
        END_EVENT
        VAR_INPUT
          QI : BOOL;
        END_VAR
      END_SUBAPPLICATION
      SUBAPPLICATION bytestringNodeIdTestRemote
        EVENT_INPUT
          INIT;
          REQ;
        END_EVENT
        EVENT_OUTPUT
          INITO;
          CNF;
        END_EVENT
        VAR_INPUT
          QI : BOOL;
        END_VAR
      END_SUBAPPLICATION
      SUBAPPLICATION stringNodeIdTestRemote
        EVENT_INPUT
          INIT;
          REQ;
        END_EVENT
        EVENT_OUTPUT
          INITO;
          CNF;
        END_EVENT
        VAR_INPUT
          QI : BOOL;
        END_VAR
      END_SUBAPPLICATION
      SUBAPPLICATION folderTestRemote
        EVENT_INPUT
          INIT;
          REQ;
        END_EVENT
        EVENT_OUTPUT
          INITO;
          CNF;
        END_EVENT
        VAR_INPUT
          QI : BOOL;
        END_VAR
      END_SUBAPPLICATION
      EVENT_CONNECTIONS
        RemoteMethods.INITO TO HandleInit.InitFinished;
        InitFinishedSignal.INITO TO PUBLISH_0.INIT;
        InitFinishedSignal.IND TO PUBLISH_0.REQ;
        bytestringNodeIdTestRemote.INITO TO RemoteMethods.INIT;
        bytestringNodeIdTestRemote.CNF TO RemoteMethods.REQ;
        HandleInit.Execute TO E_DELAY.START;
        numericNodeIdTestRemote.INITO TO stringNodeIdTestRemote.INIT;
        numericNodeIdTestRemote.CNF TO stringNodeIdTestRemote.REQ;
        stringNodeIdTestRemote.INITO TO bytestringNodeIdTestRemote.INIT;
        stringNodeIdTestRemote.CNF TO bytestringNodeIdTestRemote.REQ;
        E_PERMIT.EO TO E_SR_1.S;
        RemoteMethods.CNF TO E_SR_1.R;
        PUBLISH_0.CNF TO E_SR_2.S;
        E_SR_2.EO TO E_PERMIT.EI;
        E_SR_1.EO TO folderTestRemote.INIT;
        E_DELAY.EO TO folderTestRemote.REQ;
        folderTestRemote.INITO TO numericNodeIdTestRemote.INIT;
        folderTestRemote.CNF TO numericNodeIdTestRemote.REQ;
        START.COLD TO InitFinishedSignal.INIT;
        START.WARM TO InitFinishedSignal.INIT;
      END_CONNECTIONS
      DATA_CONNECTIONS
        E_SR_1.Q TO RemoteMethods.QI;
        E_SR_1.Q TO bytestringNodeIdTestRemote.QI;
        E_SR_1.Q TO stringNodeIdTestRemote.QI;
        E_SR_1.Q TO numericNodeIdTestRemote.QI;
        E_SR_2.Q TO E_PERMIT.PERMIT;
        E_SR_1.Q TO folderTestRemote.QI;
        E_SR_1.Q TO HandleInit.QI;
      END_CONNECTIONS
    END_RESOURCE
    RESOURCE typesClient : EMB_RES
      FBS
        RemoteRead : CLIENT_0_21(ID := opc_ua[READ;%serverEndpoint%;%opcuaTypeAll%]);
        RemoteCall : CLIENT_21(ID := opc_ua[%callMethodAction%;%serverEndpoint%;%opcuaTypeNode%]);
        E_SR_1 : E_SR;
        InitFinishedSignal : SUBSCRIBE_0(QI := 1, ID := %serverInitCommId%);
        E_PERMIT : E_PERMIT;
        E_SR_2 : E_SR;
        PUBLISH_0 : PUBLISH_0(QI := 1, ID := %serverInitCommIdACK%);
        RemoteWrite : CLIENT_21_0(ID := opc_ua[WRITE;%serverEndpoint%;%opcuaTypeAll%]);
        RemoteWriteAll : TEST_CONDITION;
      END_FBS
      SUBAPPLICATION SubApp_2
        EVENT_INPUT
          REQ;
        END_EVENT
        EVENT_OUTPUT
          CNF;
        END_EVENT
        VAR_OUTPUT
          BOOL_O : BOOL;
          SINT_O : SINT;
          INT_O : INT;
          DINT_O : DINT;
          LINT_O : LINT;
          USINT_O : USINT;
          UINT_O : UINT;
          UDINT_O : UDINT;
          ULINT_O : ULINT;
          BYTE_O : BYTE;
          WORD_O : WORD;
          DWORD_O : DWORD;
          LWORD_O : LWORD;
          DATE_O : BOOL;
          DATE_TIME_O : BOOL;
          TIME_OF_DAY_O : BOOL;
          TIME_O : TIME;
          REAL_O : REAL;
          LREAL_O : LREAL;
          STRING_O : STRING;
          WSTRING_O : WSTRING;
        END_VAR
      END_SUBAPPLICATION
      SUBAPPLICATION TypeTest_3
        EVENT_INPUT
          REQ;
        END_EVENT
        EVENT_OUTPUT
          CNF;
        END_EVENT
        VAR_INPUT
          BOOL_I : BOOL; (* BOOL Type Input *)
          SINT_I : SINT; (* SINT Type Input *)
          INT_I : INT; (* INT Type Input *)
          DINT_I : DINT; (* DINT Type Input *)
          LINT_I : LINT; (* LINT Type Input *)
          USINT_I : USINT; (* USINT Type Input *)
          UINT_I : UINT; (* UINT Type Input *)
          UDINT_I : UDINT; (* UDINT Type Input *)
          ULINT_I : ULINT; (* ULINT Type Input *)
          BYTE_I : BYTE; (* BYTE Type Input *)
          WORD_I : WORD; (* WORD Type Input *)
          DWORD_I : DWORD; (* DWORD Type Input *)
          LWORD_I : LWORD; (* LWORD Type Input *)
          DATE_I : DATE; (* DATE Type Input *)
          TIME_OF_DAY_I : TIME_OF_DAY; (* TIME_OF_DAY Type Input *)
          DATE_AND_TIME_I : DATE_AND_TIME; (* DATE_AND_TIME Type Input *)
          TIME_I : TIME; (* TIME Type Input *)
          REAL_I : REAL; (* REAL Type Input *)
          LREAL_I : LREAL; (* LREAL Type Input *)
          STRING_I : STRING; (* STRING Type Input *)
          WSTRING_I : WSTRING; (* WSTRING Type Input *)
        END_VAR
      END_SUBAPPLICATION
      SUBAPPLICATION AllTypes_2
        EVENT_INPUT
          REQ;
        END_EVENT
        EVENT_OUTPUT
          CNF;
        END_EVENT
        VAR_INPUT
          BOOL_I : BOOL; (* BOOL Type Input *)
          SINT_I : SINT; (* SINT Type Input *)
          INT_I : INT; (* INT Type Input *)
          DINT_I : DINT; (* DINT Type Input *)
          LINT_I : LINT; (* LINT Type Input *)
          USINT_I : USINT; (* USINT Type Input *)
          UINT_I : UINT; (* UINT Type Input *)
          UDINT_I : UDINT; (* UDINT Type Input *)
          ULINT_I : ULINT; (* ULINT Type Input *)
          BYTE_I : BYTE; (* BYTE Type Input *)
          WORD_I : WORD; (* WORD Type Input *)
          DWORD_I : DWORD; (* DWORD Type Input *)
          LWORD_I : LWORD; (* LWORD Type Input *)
          DATE_I_BOOL : BOOL; (* DATE Type Input *)
          TIME_OF_DAY_I_BOOL : BOOL; (* TIME_OF_DAY Type Input *)
          DATE_AND_TIME_I_BOOL : BOOL; (* DATE_AND_TIME Type Input *)
          TIME_I : TIME; (* TIME Type Input *)
          REAL_I : REAL; (* REAL Type Input *)
          LREAL_I : LREAL; (* LREAL Type Input *)
          STRING_I : STRING; (* STRING Type Input *)
          WSTRING_I : WSTRING; (* WSTRING Type Input *)
        END_VAR
        VAR_OUTPUT
          BOOL_O : BOOL; (* BOOL Type Output *)
          SINT_O : SINT; (* SINT Type Output *)
          INT_O : INT; (* INT Type Output *)
          DINT_O : DINT; (* DINT Type Output *)
          LINT_O : LINT; (* LINT Type Output *)
          USINT_O : USINT; (* USINT Type Output *)
          UINT_O : UINT; (* UINT Type Output *)
          UDINT_O : UDINT; (* UDINT Type Output *)
          ULINT_O : ULINT; (* ULINT Type Output *)
          BYTE_O : BYTE; (* BYTE Type Output *)
          WORD_O : WORD; (* WORD Type Output *)
          DWORD_O : DWORD; (* DWORD Type Output *)
          LWORD_O : LWORD; (* LWORD Type Output *)
          DATE_O_BOOL : BOOL; (* DATE Type Output *)
          TIME_OF_DAY_O_BOOL : BOOL; (* TIME_OF_DAY Type Output *)
          DATE_AND_TIME_O_BOOL : BOOL; (* DATE_AND_TIME Type Output *)
          TIME_O : TIME; (* TIME Type Output *)
          REAL_O : REAL; (* REAL Type Output *)
          LREAL_O : LREAL; (* LREAL Type Output *)
          STRING_O : STRING; (* STRING Type Output *)
          WSTRING_O : WSTRING; (* WSTRING Type Output *)
        END_VAR
      END_SUBAPPLICATION
      SUBAPPLICATION AllTypes_3
        EVENT_INPUT
          REQ;
        END_EVENT
        EVENT_OUTPUT
          CNF;
        END_EVENT
        VAR_INPUT
          BOOL_I : BOOL; (* BOOL Type Input *)
          SINT_I : SINT; (* SINT Type Input *)
          INT_I : INT; (* INT Type Input *)
          DINT_I : DINT; (* DINT Type Input *)
          LINT_I : LINT; (* LINT Type Input *)
          USINT_I : USINT; (* USINT Type Input *)
          UINT_I : UINT; (* UINT Type Input *)
          UDINT_I : UDINT; (* UDINT Type Input *)
          ULINT_I : ULINT; (* ULINT Type Input *)
          BYTE_I : BYTE; (* BYTE Type Input *)
          WORD_I : WORD; (* WORD Type Input *)
          DWORD_I : DWORD; (* DWORD Type Input *)
          LWORD_I : LWORD; (* LWORD Type Input *)
          DATE_I_BOOL : BOOL; (* DATE Type Input *)
          TIME_OF_DAY_I_BOOL : BOOL; (* TIME_OF_DAY Type Input *)
          DATE_AND_TIME_I_BOOL : BOOL; (* DATE_AND_TIME Type Input *)
          TIME_I : TIME; (* TIME Type Input *)
          REAL_I : REAL; (* REAL Type Input *)
          LREAL_I : LREAL; (* LREAL Type Input *)
          STRING_I : STRING; (* STRING Type Input *)
          WSTRING_I : WSTRING; (* WSTRING Type Input *)
        END_VAR
        VAR_OUTPUT
          BOOL_O : BOOL; (* BOOL Type Output *)
          SINT_O : SINT; (* SINT Type Output *)
          INT_O : INT; (* INT Type Output *)
          DINT_O : DINT; (* DINT Type Output *)
          LINT_O : LINT; (* LINT Type Output *)
          USINT_O : USINT; (* USINT Type Output *)
          UINT_O : UINT; (* UINT Type Output *)
          UDINT_O : UDINT; (* UDINT Type Output *)
          ULINT_O : ULINT; (* ULINT Type Output *)
          BYTE_O : BYTE; (* BYTE Type Output *)
          WORD_O : WORD; (* WORD Type Output *)
          DWORD_O : DWORD; (* DWORD Type Output *)
          LWORD_O : LWORD; (* LWORD Type Output *)
          DATE_O_BOOL : BOOL; (* DATE Type Output *)
          TIME_OF_DAY_O_BOOL : BOOL; (* TIME_OF_DAY Type Output *)
          DATE_AND_TIME_O_BOOL : BOOL; (* DATE_AND_TIME Type Output *)
          TIME_O : TIME; (* TIME Type Output *)
          REAL_O : REAL; (* REAL Type Output *)
          LREAL_O : LREAL; (* LREAL Type Output *)
          STRING_O : STRING; (* STRING Type Output *)
          WSTRING_O : WSTRING; (* WSTRING Type Output *)
        END_VAR
      END_SUBAPPLICATION
      SUBAPPLICATION TypeTest_2
        EVENT_INPUT
          REQ;
        END_EVENT
        EVENT_OUTPUT
          CNF;
        END_EVENT
        VAR_INPUT
          BOOL_I : BOOL; (* BOOL Type Input *)
          SINT_I : SINT; (* SINT Type Input *)
          INT_I : INT; (* INT Type Input *)
          DINT_I : DINT; (* DINT Type Input *)
          LINT_I : LINT; (* LINT Type Input *)
          USINT_I : USINT; (* USINT Type Input *)
          UINT_I : UINT; (* UINT Type Input *)
          UDINT_I : UDINT; (* UDINT Type Input *)
          ULINT_I : ULINT; (* ULINT Type Input *)
          BYTE_I : BYTE; (* BYTE Type Input *)
          WORD_I : WORD; (* WORD Type Input *)
          DWORD_I : DWORD; (* DWORD Type Input *)
          LWORD_I : LWORD; (* LWORD Type Input *)
          DATE_I : DATE; (* DATE Type Input *)
          TIME_OF_DAY_I : TIME_OF_DAY; (* TIME_OF_DAY Type Input *)
          DATE_AND_TIME_I : DATE_AND_TIME; (* DATE_AND_TIME Type Input *)
          TIME_I : TIME; (* TIME Type Input *)
          REAL_I : REAL; (* REAL Type Input *)
          LREAL_I : LREAL; (* LREAL Type Input *)
          STRING_I : STRING; (* STRING Type Input *)
          WSTRING_I : WSTRING; (* WSTRING Type Input *)
        END_VAR
      END_SUBAPPLICATION
      SUBAPPLICATION HandleInit
        EVENT_INPUT
          InitFinished;
        END_EVENT
        EVENT_OUTPUT
          Execute;
        END_EVENT
        VAR_INPUT
          QI : BOOL;
        END_VAR
      END_SUBAPPLICATION
      SUBAPPLICATION SubApp
        EVENT_INPUT
          REQ;
        END_EVENT
        EVENT_OUTPUT
          CNF;
        END_EVENT
        VAR_OUTPUT
          BOOL_O : BOOL;
          SINT_O : SINT;
          INT_O : INT;
          DINT_O : DINT;
          LINT_O : LINT;
          USINT_O : USINT;
          UINT_O : UINT;
          UDINT_O : UDINT;
          ULINT_O : ULINT;
          BYTE_O : BYTE;
          WORD_o : WORD;
          DWORD_O : DWORD;
          LWORD_O : LWORD;
          DATE_O : BOOL;
          DATE_TIME_O : BOOL;
          TIME_OF_DAY_O : BOOL;
          TIME_O : TIME;
          REAL_O : REAL;
          LREAL_O : LREAL;
          STRING_O : STRING;
          WSTRING_O : WSTRING;
        END_VAR
      END_SUBAPPLICATION
      EVENT_CONNECTIONS
        RemoteRead.CNF TO AllTypes_2.REQ;
        RemoteRead.INITO TO RemoteCall.INIT;
        SubApp_2.CNF TO RemoteCall.REQ;
        RemoteCall.CNF TO AllTypes_3.REQ;
        AllTypes_3.CNF TO TypeTest_3.REQ;
        AllTypes_2.CNF TO TypeTest_2.REQ;
        TypeTest_2.CNF TO SubApp_2.REQ;
        RemoteCall.INITO TO HandleInit.InitFinished;
        TypeTest_3.CNF TO E_SR_1.R;
        E_PERMIT.EO TO E_SR_1.S;
        HandleInit.Execute TO SubApp.REQ;
        E_SR_2.EO TO E_PERMIT.EI;
        InitFinishedSignal.INITO TO PUBLISH_0.INIT;
        InitFinishedSignal.IND TO PUBLISH_0.REQ;
        PUBLISH_0.CNF TO E_SR_2.S;
        START.COLD TO InitFinishedSignal.INIT;
        START.WARM TO InitFinishedSignal.INIT;
        E_SR_1.EO TO RemoteWrite.INIT;
        SubApp.CNF TO RemoteWrite.REQ;
        RemoteWrite.INITO TO RemoteRead.INIT;
        RemoteWrite.CNF TO RemoteWriteAll.REQ;
        RemoteWriteAll.CNF TO RemoteRead.REQ;
      END_CONNECTIONS
      DATA_CONNECTIONS
        RemoteRead.RD_1 TO AllTypes_2.BOOL_I;
        RemoteRead.RD_2 TO AllTypes_2.SINT_I;
        RemoteRead.RD_3 TO AllTypes_2.INT_I;
        RemoteRead.RD_4 TO AllTypes_2.DINT_I;
        RemoteRead.RD_5 TO AllTypes_2.LINT_I;
        RemoteRead.RD_6 TO AllTypes_2.USINT_I;
        RemoteRead.RD_7 TO AllTypes_2.UINT_I;
        RemoteRead.RD_8 TO AllTypes_2.UDINT_I;
        RemoteRead.RD_9 TO AllTypes_2.ULINT_I;
        RemoteRead.RD_10 TO AllTypes_2.BYTE_I;
        RemoteRead.RD_11 TO AllTypes_2.WORD_I;
        RemoteRead.RD_12 TO AllTypes_2.DWORD_I;
        RemoteRead.RD_13 TO AllTypes_2.LWORD_I;
        RemoteRead.RD_14 TO AllTypes_2.DATE_I_BOOL;
        RemoteRead.RD_15 TO AllTypes_2.TIME_OF_DAY_I_BOOL;
        RemoteRead.RD_16 TO AllTypes_2.DATE_AND_TIME_I_BOOL;
        RemoteRead.RD_17 TO AllTypes_2.TIME_I;
        RemoteRead.RD_18 TO AllTypes_2.REAL_I;
        RemoteRead.RD_19 TO AllTypes_2.LREAL_I;
        RemoteRead.RD_20 TO AllTypes_2.STRING_I;
        RemoteRead.RD_21 TO AllTypes_2.WSTRING_I;
        SubApp_2.BOOL_O TO RemoteCall.SD_1;
        SubApp_2.SINT_O TO RemoteCall.SD_2;
        SubApp_2.INT_O TO RemoteCall.SD_3;
        SubApp_2.DINT_O TO RemoteCall.SD_4;
        SubApp_2.LINT_O TO RemoteCall.SD_5;
        SubApp_2.USINT_O TO RemoteCall.SD_6;
        SubApp_2.UINT_O TO RemoteCall.SD_7;
        SubApp_2.UDINT_O TO RemoteCall.SD_8;
        SubApp_2.ULINT_O TO RemoteCall.SD_9;
        SubApp_2.BYTE_O TO RemoteCall.SD_10;
        SubApp_2.WORD_O TO RemoteCall.SD_11;
        SubApp_2.DWORD_O TO RemoteCall.SD_12;
        SubApp_2.LWORD_O TO RemoteCall.SD_13;
        SubApp_2.DATE_O TO RemoteCall.SD_14;
        SubApp_2.DATE_TIME_O TO RemoteCall.SD_15;
        SubApp_2.TIME_OF_DAY_O TO RemoteCall.SD_16;
        SubApp_2.TIME_O TO RemoteCall.SD_17;
        SubApp_2.REAL_O TO RemoteCall.SD_18;
        SubApp_2.LREAL_O TO RemoteCall.SD_19;
        SubApp_2.STRING_O TO RemoteCall.SD_20;
        SubApp_2.WSTRING_O TO RemoteCall.SD_21;
        RemoteCall.RD_1 TO AllTypes_3.BOOL_I;
        RemoteCall.RD_2 TO AllTypes_3.SINT_I;
        RemoteCall.RD_3 TO AllTypes_3.INT_I;
        RemoteCall.RD_4 TO AllTypes_3.DINT_I;
        RemoteCall.RD_5 TO AllTypes_3.LINT_I;
        RemoteCall.RD_6 TO AllTypes_3.USINT_I;
        RemoteCall.RD_7 TO AllTypes_3.UINT_I;
        RemoteCall.RD_8 TO AllTypes_3.UDINT_I;
        RemoteCall.RD_9 TO AllTypes_3.ULINT_I;
        RemoteCall.RD_10 TO AllTypes_3.BYTE_I;
        RemoteCall.RD_11 TO AllTypes_3.WORD_I;
        RemoteCall.RD_12 TO AllTypes_3.DWORD_I;
        RemoteCall.RD_13 TO AllTypes_3.LWORD_I;
        RemoteCall.RD_14 TO AllTypes_3.DATE_I_BOOL;
        RemoteCall.RD_15 TO AllTypes_3.TIME_OF_DAY_I_BOOL;
        RemoteCall.RD_16 TO AllTypes_3.DATE_AND_TIME_I_BOOL;
        RemoteCall.RD_17 TO AllTypes_3.TIME_I;
        RemoteCall.RD_18 TO AllTypes_3.REAL_I;
        RemoteCall.RD_19 TO AllTypes_3.LREAL_I;
        RemoteCall.RD_20 TO AllTypes_3.STRING_I;
        RemoteCall.RD_21 TO AllTypes_3.WSTRING_I;
        AllTypes_3.BOOL_O TO TypeTest_3.BOOL_I;
        AllTypes_3.SINT_O TO TypeTest_3.SINT_I;
        AllTypes_3.INT_O TO TypeTest_3.INT_I;
        AllTypes_3.DINT_O TO TypeTest_3.DINT_I;
        AllTypes_3.LINT_O TO TypeTest_3.LINT_I;
        AllTypes_3.USINT_O TO TypeTest_3.USINT_I;
        AllTypes_3.UINT_O TO TypeTest_3.UINT_I;
        AllTypes_3.UDINT_O TO TypeTest_3.UDINT_I;
        AllTypes_3.ULINT_O TO TypeTest_3.ULINT_I;
        AllTypes_3.BYTE_O TO TypeTest_3.BYTE_I;
        AllTypes_3.WORD_O TO TypeTest_3.WORD_I;
        AllTypes_3.DWORD_O TO TypeTest_3.DWORD_I;
        AllTypes_3.LWORD_O TO TypeTest_3.LWORD_I;
        AllTypes_3.DATE_O_BOOL TO TypeTest_3.DATE_I;
        AllTypes_3.TIME_OF_DAY_O_BOOL TO TypeTest_3.TIME_OF_DAY_I;
        AllTypes_3.DATE_AND_TIME_O_BOOL TO TypeTest_3.DATE_AND_TIME_I;
        AllTypes_3.TIME_O TO TypeTest_3.TIME_I;
        AllTypes_3.REAL_O TO TypeTest_3.REAL_I;
        AllTypes_3.LREAL_O TO TypeTest_3.LREAL_I;
        AllTypes_3.STRING_O TO TypeTest_3.STRING_I;
        AllTypes_3.WSTRING_O TO TypeTest_3.WSTRING_I;
        AllTypes_2.BOOL_O TO TypeTest_2.BOOL_I;
        AllTypes_2.SINT_O TO TypeTest_2.SINT_I;
        AllTypes_2.INT_O TO TypeTest_2.INT_I;
        AllTypes_2.DINT_O TO TypeTest_2.DINT_I;
        AllTypes_2.LINT_O TO TypeTest_2.LINT_I;
        AllTypes_2.USINT_O TO TypeTest_2.USINT_I;
        AllTypes_2.UINT_O TO TypeTest_2.UINT_I;
        AllTypes_2.UDINT_O TO TypeTest_2.UDINT_I;
        AllTypes_2.ULINT_O TO TypeTest_2.ULINT_I;
        AllTypes_2.BYTE_O TO TypeTest_2.BYTE_I;
        AllTypes_2.WORD_O TO TypeTest_2.WORD_I;
        AllTypes_2.DWORD_O TO TypeTest_2.DWORD_I;
        AllTypes_2.LWORD_O TO TypeTest_2.LWORD_I;
        AllTypes_2.DATE_O_BOOL TO TypeTest_2.DATE_I;
        AllTypes_2.TIME_OF_DAY_O_BOOL TO TypeTest_2.TIME_OF_DAY_I;
        AllTypes_2.DATE_AND_TIME_O_BOOL TO TypeTest_2.DATE_AND_TIME_I;
        AllTypes_2.TIME_O TO TypeTest_2.TIME_I;
        AllTypes_2.REAL_O TO TypeTest_2.REAL_I;
        AllTypes_2.LREAL_O TO TypeTest_2.LREAL_I;
        AllTypes_2.STRING_O TO TypeTest_2.STRING_I;
        AllTypes_2.WSTRING_O TO TypeTest_2.WSTRING_I;
        E_SR_1.Q TO HandleInit.QI;
        E_SR_1.Q TO RemoteRead.QI;
        E_SR_1.Q TO RemoteCall.QI;
        E_SR_2.Q TO E_PERMIT.PERMIT;
        E_SR_1.Q TO RemoteWrite.QI;
        SubApp.BOOL_O TO RemoteWrite.SD_1;
        SubApp.SINT_O TO RemoteWrite.SD_2;
        SubApp.INT_O TO RemoteWrite.SD_3;
        SubApp.DINT_O TO RemoteWrite.SD_4;
        SubApp.LINT_O TO RemoteWrite.SD_5;
        SubApp.USINT_O TO RemoteWrite.SD_6;
        SubApp.UINT_O TO RemoteWrite.SD_7;
        SubApp.UDINT_O TO RemoteWrite.SD_8;
        SubApp.ULINT_O TO RemoteWrite.SD_9;
        SubApp.BYTE_O TO RemoteWrite.SD_10;
        SubApp.WORD_o TO RemoteWrite.SD_11;
        SubApp.DWORD_O TO RemoteWrite.SD_12;
        SubApp.LWORD_O TO RemoteWrite.SD_13;
        SubApp.DATE_O TO RemoteWrite.SD_14;
        SubApp.DATE_TIME_O TO RemoteWrite.SD_15;
        SubApp.TIME_OF_DAY_O TO RemoteWrite.SD_16;
        SubApp.TIME_O TO RemoteWrite.SD_17;
        SubApp.REAL_O TO RemoteWrite.SD_18;
        SubApp.LREAL_O TO RemoteWrite.SD_19;
        SubApp.STRING_O TO RemoteWrite.SD_20;
        SubApp.WSTRING_O TO RemoteWrite.SD_21;
        RemoteWrite.QO TO RemoteWriteAll.check;
      END_CONNECTIONS
    END_RESOURCE
    RESOURCE testClient : EMB_RES
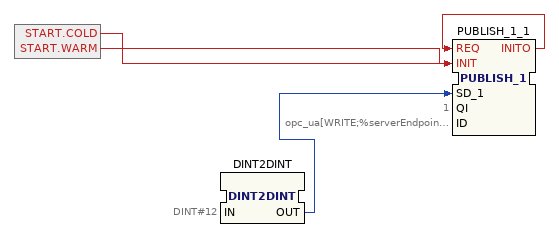
      FBS
        PUBLISH_1_1 : PUBLISH_1(QI := 1, ID := opc_ua[WRITE;%serverEndpoint%;%opcuaWRITEVariable%]);
        DINT2DINT : DINT2DINT(IN := DINT#12);
      END_FBS
      EVENT_CONNECTIONS
        PUBLISH_1_1.INITO TO PUBLISH_1_1.REQ;
        START.COLD TO PUBLISH_1_1.INIT;
        START.WARM TO PUBLISH_1_1.INIT;
      END_CONNECTIONS
      DATA_CONNECTIONS
        DINT2DINT.OUT TO PUBLISH_1_1.SD_1;
      END_CONNECTIONS
    END_RESOURCE
  END_DEVICE
  MAPPINGS
    OpcUWrongParameters.STEST_END ON OPCUAServer.WrongParameters.STEST_END;
    OpcUWrongParameters.NoSemicolon ON OPCUAServer.WrongParameters.NoSemicolon;
    OpcUWrongParameters.W2W ON OPCUAServer.WrongParameters.W2W;
    OpcUWrongParameters.W2W_1 ON OPCUAServer.WrongParameters.W2W_1;
    OpcUWrongParameters.emptyAction ON OPCUAServer.WrongParameters.emptyAction;
    OpcUWrongParameters.W2W_1_1 ON OPCUAServer.WrongParameters.W2W_1_1;
    OpcUWrongParameters.NoExistingAction ON OPCUAServer.WrongParameters.NoExistingAction;
    OpcUWrongParameters.UnknownIdentifier ON OPCUAServer.WrongParameters.UnknownIdentifier;
    OpcUWrongParameters.W2W_1_1_1 ON OPCUAServer.WrongParameters.W2W_1_1_1;
    OpcUWrongParameters.WrongIdentifier ON OPCUAServer.WrongParameters.WrongIdentifier;
    OpcUWrongParameters.W2W_1_1_4 ON OPCUAServer.WrongParameters.W2W_1_1_4;
    OpcUWrongParameters.W2W_1_1_2 ON OPCUAServer.WrongParameters.W2W_1_1_2;
    OpcUWrongParameters.W2W_1_1_3 ON OPCUAServer.WrongParameters.W2W_1_1_3;
    OpcUWrongParameters.wrongNodeId ON OPCUAServer.WrongParameters.wrongNodeId;
    OpcUWrongParameters.wrongPair ON OPCUAServer.WrongParameters.wrongPair;
    OpcUWrongParameters.LocalWithoutBrowseName ON OPCUAServer.WrongParameters.LocalWithoutBrowseName;
    OpcUWrongParameters.RemoteWithoutBrowseNameNorNodeId ON OPCUAServer.WrongParameters.RemoteWithoutBrowseNameNorNodeId;
    OpcUWrongParameters.W2W_1_1_4_1 ON OPCUAServer.WrongParameters.W2W_1_1_4_1;
    OpcUWrongParameters.W2W_1_1_4_2 ON OPCUAServer.WrongParameters.W2W_1_1_4_2;
    OpcUWrongParameters.RemoteRead ON OPCUAServer.WrongParameters.RemoteRead;
    OpcUWrongParameters.W2W_1_1_4_2_1_1 ON OPCUAServer.WrongParameters.W2W_1_1_4_2_1_1;
    OpcUWrongParameters.LocalRead ON OPCUAServer.WrongParameters.LocalRead;
    OpcUWrongParameters.W2W_1_1_4_2_1 ON OPCUAServer.WrongParameters.W2W_1_1_4_2_1;
    OpcUWrongParameters.W2W_1_1_4_2_1_1_1 ON OPCUAServer.WrongParameters.W2W_1_1_4_2_1_1_1;
    OpcUWrongParameters.RemoteWrite ON OPCUAServer.WrongParameters.RemoteWrite;
    OpcUWrongParameters.W2W_1_1_4_2_1_1_1_1 ON OPCUAServer.WrongParameters.W2W_1_1_4_2_1_1_1_1;
    OpcUWrongParameters.LocalWrite ON OPCUAServer.WrongParameters.LocalWrite;
    OpcUWrongParameters.CreateMethod ON OPCUAServer.WrongParameters.CreateMethod;
    OpcUWrongParameters.W2W_1_1_4_2_1_1_1_1_1 ON OPCUAServer.WrongParameters.W2W_1_1_4_2_1_1_1_1_1;
    OpcUWrongParameters.CallMethod ON OPCUAServer.WrongParameters.CallMethod;
    OpcUWrongParameters.W2W_1_1_4_2_1_1_1_1_1_1 ON OPCUAServer.WrongParameters.W2W_1_1_4_2_1_1_1_1_1_1;
    OpcUWrongParameters.Subscribe ON OPCUAServer.WrongParameters.Subscribe;
    OpcUWrongParameters.W2W_1_1_4_2_1_1_1_1_1_1_1 ON OPCUAServer.WrongParameters.W2W_1_1_4_2_1_1_1_1_1_1_1;
    OpcUaLocalWorking.E_SR ON OPCUAServer.foldersReadFirst.E_SR;
    OpcUaLocalWorking.FoldersNoBrowseName ON OPCUAServer.foldersReadFirst.FoldersNoBrowseName;
    OpcUaLocalWorking.foldersWithNodeStringId ON OPCUAServer.foldersReadFirst.foldersWithNodeStringId;
    OpcUaLocalWorking.foldersWithNodeNumericId ON OPCUAServer.foldersReadFirst.foldersWithNodeNumericId;
    OpcUaLocalWorking.foldersWithNodeByteStringId ON OPCUAServer.foldersReadFirst.foldersWithNodeByteStringId;
    OpcUaLocalWorking.STEST_END ON OPCUAServer.foldersReadFirst.STEST_END;
    OpcUaLocalWorking.E_DEMUX_2 ON OPCUAServer.foldersReadFirst.E_DEMUX_2;
    OpcUaLocalWorking.F_BOOL_TO_UINT ON OPCUAServer.foldersReadFirst.F_BOOL_TO_UINT;
    OpcUaLocalWorking.STEST_END_1 ON OPCUAServer.foldersWriteFirst.STEST_END_1;
    OpcUaLocalWorking.FoldersNoBrowseName_1 ON OPCUAServer.foldersWriteFirst.FoldersNoBrowseName_1;
    OpcUaLocalWorking.foldersWithNodeByteStringId_1 ON OPCUAServer.foldersWriteFirst.foldersWithNodeByteStringId_1;
    OpcUaLocalWorking.foldersWithNodeNumericId_1 ON OPCUAServer.foldersWriteFirst.foldersWithNodeNumericId_1;
    OpcUaLocalWorking.F_BOOL_TO_UINT_1 ON OPCUAServer.foldersWriteFirst.F_BOOL_TO_UINT_1;
    OpcUaLocalWorking.foldersWithNodeStringId_1 ON OPCUAServer.foldersWriteFirst.foldersWithNodeStringId_1;
    OpcUaLocalWorking.E_DEMUX_2_1 ON OPCUAServer.foldersWriteFirst.E_DEMUX_2_1;
    OpcUaLocalWorking.E_SR_1 ON OPCUAServer.foldersWriteFirst.E_SR_1;
    OpcUaLocalWorking.F_BOOL_TO_UINT_2 ON OPCUAServer.createLocalMethods.F_BOOL_TO_UINT_2;
    OpcUaLocalWorking.MethodOnlyBrowseName ON OPCUAServer.createLocalMethods.MethodOnlyBrowseName;
    OpcUaLocalWorking.MethodBytestringNodeId ON OPCUAServer.createLocalMethods.MethodBytestringNodeId;
    OpcUaLocalWorking.E_DEMUX_2_2 ON OPCUAServer.createLocalMethods.E_DEMUX_2_2;
    OpcUaLocalWorking.E_SR_2 ON OPCUAServer.createLocalMethods.E_SR_2;
    OpcUaLocalWorking.MethodNumericNodeId ON OPCUAServer.createLocalMethods.MethodNumericNodeId;
    OpcUaLocalWorking.MethodStringNodeId ON OPCUAServer.createLocalMethods.MethodStringNodeId;
    OpcUaLocalWorking.STEST_END_2 ON OPCUAServer.createLocalMethods.STEST_END_2;
    OpcUaBothWorking.E_SR ON OPCUAServer.WorkingServer.E_SR;
    OpcUaBothWorking.E_SR_1 ON OPCUACLient.WorkingClient.E_SR_1;
    OpcUaBothWorking.InitFinishedSignal ON OPCUACLient.WorkingClient.InitFinishedSignal;
    OpcUaBothWorking.SUBSCRIBE_0_1 ON OPCUAServer.WorkingServer.SUBSCRIBE_0_1;
    OpcUaBothWorking.folderTest ON OPCUAServer.WorkingServer.folderTest;
    OpcUaBothWorking.PUBLISH_0 ON OPCUACLient.WorkingClient.PUBLISH_0;
    OpcUaBothWorking.folderTestRemote ON OPCUACLient.WorkingClient.folderTestRemote;
    OpcUaBothWorking.HandleInit ON OPCUACLient.WorkingClient.HandleInit;
    OpcUaBothWorking.HandleInitLocal ON OPCUAServer.WorkingServer.HandleInitLocal;
    OpcUaBothWorking.numericNodeIdTestRemote ON OPCUACLient.WorkingClient.numericNodeIdTestRemote;
    OpcUaBothWorking.stringNodeIdTestRemote ON OPCUACLient.WorkingClient.stringNodeIdTestRemote;
    OpcUaBothWorking.bytestringNodeIdTestRemote ON OPCUACLient.WorkingClient.bytestringNodeIdTestRemote;
    OpcUaBothWorking.E_SR_2 ON OPCUACLient.WorkingClient.E_SR_2;
    OpcUaBothWorking.E_PERMIT ON OPCUACLient.WorkingClient.E_PERMIT;
    OpcUaBothWorking.E_DELAY ON OPCUACLient.WorkingClient.E_DELAY;
    OpcUWrongParameters.W2W_2 ON OPCUAServer.WrongParameters.W2W_2;
    OpcUWrongParameters.GUIDIdentifier ON OPCUAServer.WrongParameters.GUIDIdentifier;
    OpcUaBothWorking.LocaMethods ON OPCUAServer.WorkingServer.LocaMethods;
    OpcUaBothWorking.RemoteMethods ON OPCUACLient.WorkingClient.RemoteMethods;
    OpcUaBothFailingCases.E_SWITCH_1 ON OPCUACLient.FailingClient.E_SWITCH_1;
    OpcUaBothFailingCases.InitFinishedSignal ON OPCUACLient.FailingClient.InitFinishedSignal;
    OpcUaBothFailingCases.HandleInit ON OPCUACLient.FailingClient.HandleInit;
    OpcUaBothFailingCases.E_DELAY ON OPCUACLient.FailingClient.E_DELAY;
    OpcUaBothFailingCases.E_SR_2 ON OPCUACLient.FailingClient.E_SR_2;
    OpcUaBothFailingCases.PUBLISH_0 ON OPCUACLient.FailingClient.PUBLISH_0;
    OpcUaBothFailingCases.E_SWITCH ON OPCUAServer.FailingServer.E_SWITCH;
    OpcUaBothFailingCases.WorngInputs ON OPCUAServer.FailingServer.WorngInputs;
    OpcUaBothFailingCases.E_SR ON OPCUAServer.FailingServer.E_SR;
    OpcUaBothFailingCases.GoodInputs ON OPCUAServer.FailingServer.GoodInputs;
    OpcUaBothFailingCases.SUBSCRIBE_0_1 ON OPCUAServer.FailingServer.SUBSCRIBE_0_1;
    OpcUaBothFailingCases.WorngInputsOutputs ON OPCUAServer.FailingServer.WorngInputsOutputs;
    OpcUaBothFailingCases.HandleInitLocal ON OPCUAServer.FailingServer.HandleInitLocal;
    OpcUaBothFailingCases.UnknownNode ON OPCUACLient.FailingClient.UnknownNode;
    OpcUaBothFailingCases.WrongNoOfArguments ON OPCUACLient.FailingClient.WrongNoOfArguments;
    OpcUaBothFailingCases.Writable1 ON OPCUAServer.FailingServer.Writable1;
    OpcUaBothFailingCases.WorngInputsType ON OPCUAServer.FailingServer.WorngInputsType;
    OpcUaBothFailingCases.BOOL2BOOL_2_1 ON OPCUAServer.FailingServer.BOOL2BOOL_2_1;
    OpcUaBothFailingCases.WrongType ON OPCUACLient.FailingClient.WrongType;
    OpcUaBothFailingCases.SERVER_0 ON OPCUAServer.FailingServer.SERVER_0;
    OpcUaBothFailingCases.SERVER_0_1 ON OPCUAServer.FailingServer.SERVER_0_1;
    OpcUaBothFailingCases.SERVER_0_1_1 ON OPCUAServer.FailingServer.SERVER_0_1_1;
    OpcUaBothFailingCases.DINT2DINT ON OPCUAServer.FailingServer.DINT2DINT;
    OpcUaBothFailingCases.DINT2DINT_1_1 ON OPCUAServer.FailingServer.DINT2DINT_1_1;
    OpcUaBothFailingCases.DINT2DINT_1 ON OPCUAServer.FailingServer.DINT2DINT_1;
    OpcUaBothFailingCases.SameNodeIdWrite ON OPCUAServer.FailingServer.SameNodeIdWrite;
    OpcUaBothFailingCases.BOOL2BOOL_2_1_1 ON OPCUAServer.FailingServer.BOOL2BOOL_2_1_1;
    OpcUaBothFailingCases.Writable1_1 ON OPCUAServer.FailingServer.Writable1_1;
    OpcUaBothFailingCases.BOOL2BOOL_2_1_1_1 ON OPCUAServer.FailingServer.BOOL2BOOL_2_1_1_1;
    OpcUaBothFailingCases.SameNameDifferentNodeIdW ON OPCUAServer.FailingServer.SameNameDifferentNodeIdW;
    OpcUaBothFailingCases.Writable1_1_1 ON OPCUAServer.FailingServer.Writable1_1_1;
    OpcUaBothFailingCases.SUBSCRIBE_1_1 ON OPCUAServer.FailingServer.SUBSCRIBE_1_1;
    OpcUaBothFailingCases.BOOL2BOOL_3_1 ON OPCUAServer.FailingServer.BOOL2BOOL_3_1;
    OpcUaBothFailingCases.SUBSCRIBE_1_1_1 ON OPCUAServer.FailingServer.SUBSCRIBE_1_1_1;
    OpcUaBothFailingCases.BOOL2BOOL_3 ON OPCUAServer.FailingServer.BOOL2BOOL_3;
    OpcUaBothFailingCases.SameNodeSecondRead ON OPCUAServer.FailingServer.SameNodeSecondRead;
    OpcUaBothFailingCases.ReadExistingWritable ON OPCUAServer.FailingServer.ReadExistingWritable;
    OpcUaBothFailingCases.F_NOT_1_1 ON OPCUAServer.FailingServer.F_NOT_1_1;
    OpcUaBothFailingCases.F_NOT ON OPCUAServer.FailingServer.F_NOT;
    OpcUaBothFailingCases.SUBSCRIBE_1_1_1_1 ON OPCUAServer.FailingServer.SUBSCRIBE_1_1_1_1;
    OpcUaBothFailingCases.SUBSCRIBE_wrongPath ON OPCUAServer.FailingServer.SUBSCRIBE_wrongPath;
    OpcUaBothFailingCases.F_NOT_1_2_1_1 ON OPCUAServer.FailingServer.F_NOT_1_2_1_1;
    OpcUaBothFailingCases.SERVER_0_2 ON OPCUAServer.FailingServer.SERVER_0_2;
    OpcUaBothFailingCases.DoubleMethod ON OPCUAServer.FailingServer.DoubleMethod;
    OpcUaBothFailingCases.BOOL2BOOL_3_2 ON OPCUAServer.FailingServer.BOOL2BOOL_3_2;
    OpcUaBothFailingCases.BOOL2BOOL_3_1_1_1 ON OPCUAServer.FailingServer.BOOL2BOOL_3_1_1_1;
    OpcUaBothFailingCases.F_NOT_1_2_1 ON OPCUAServer.FailingServer.F_NOT_1_2_1;
    OpcUaBothFailingCases.ValidNode ON OPCUAServer.FailingServer.ValidNode;
    OpcUaBothFailingCases.WrongPath ON OPCUAServer.FailingServer.WrongPath;
    OpcUaBothFailingCases.BOOL2BOOL_3_1_1 ON OPCUAServer.FailingServer.BOOL2BOOL_3_1_1;
    OpcUaBothFailingCases.BOOL2BOOL_3_2_1_1 ON OPCUAServer.FailingServer.BOOL2BOOL_3_2_1_1;
    OpcUaBothFailingCases.F_NOT_1_2_1_1_1_1 ON OPCUAServer.FailingServer.F_NOT_1_2_1_1_1_1;
    OpcUaBothFailingCases.SUBSCRIBE_150 ON OPCUAServer.FailingServer.SUBSCRIBE_150;
    OpcUaBothFailingCases.UnconnectedRD ON OPCUAServer.FailingServer.UnconnectedRD;
    OpcUaBothFailingCases.UnconnectedSD ON OPCUAServer.FailingServer.UnconnectedSD;
    OpcUaBothFailingCases.BOOL2BOOL_3_2_1 ON OPCUAServer.FailingServer.BOOL2BOOL_3_2_1;
    OpcUaBothFailingCases.STRING2STRING_1 ON OPCUAServer.FailingServer.STRING2STRING_1;
    OpcUaBothFailingCases.F_NOT_1 ON OPCUAServer.FailingServer.F_NOT_1;
    OpcUaBothFailingCases.F_NOT_1_2_1_1_1 ON OPCUAServer.FailingServer.F_NOT_1_2_1_1_1;
    OpcUaBothFailingCases.DifferentTypesOutput ON OPCUAServer.FailingServer.DifferentTypesOutput;
    OpcUaBothFailingCases.SUBSCRIBE_140 ON OPCUAServer.FailingServer.SUBSCRIBE_140;
    OpcUaBothFailingCases.Writable1_1_2 ON OPCUAServer.FailingServer.Writable1_1_2;
    OpcUaBothFailingCases.SameNodeIdRead ON OPCUAServer.FailingServer.SameNodeIdRead;
    OpcUaBothFailingCases.SUBSCRIBE_1 ON OPCUAServer.FailingServer.SUBSCRIBE_1;
    OpcUaBothFailingCases.BOOL2BOOL_2_1_1_2 ON OPCUAServer.FailingServer.BOOL2BOOL_2_1_1_2;
    OpcUaBothFailingCases.F_NOT_2 ON OPCUAServer.FailingServer.F_NOT_2;
    OpcUaBothFailingCases.F_EQ ON OPCUAServer.FailingServer.F_EQ;
    OpcUaBothFailingCases.SameNameDifferentNodeIdR ON OPCUAServer.FailingServer.SameNameDifferentNodeIdR;
    OpcUaBothFailingCases.Writable1_2 ON OPCUAServer.FailingServer.Writable1_2;
    OpcUaBothFailingCases.BOOL2BOOL_3_3 ON OPCUAServer.FailingServer.BOOL2BOOL_3_3;
    OpcUaBothFailingCases.STRING2STRING ON OPCUAServer.FailingServer.STRING2STRING;
    OpcUaBothFailingCases.WrongInputOutput ON OPCUACLient.FailingClient.WrongInputOutput;
    OpcUaBothFailingCases.BOOL2BOOL_3_2_1_2 ON OPCUAServer.FailingServer.BOOL2BOOL_3_2_1_2;
    OpcUaBothFailingCases.SameTypesOutput ON OPCUAServer.FailingServer.SameTypesOutput;
    OpcUaBothFailingCases.SUBSCRIBE_150_1 ON OPCUAServer.FailingServer.SUBSCRIBE_150_1;
    OpcUaBothFailingCases.F_NOT_1_2_1_2_1 ON OPCUAServer.FailingServer.F_NOT_1_2_1_2_1;
    OpcUaBothFailingCases.F_NOT_1_2_1_2 ON OPCUAServer.FailingServer.F_NOT_1_2_1_2;
    OpcUaBothFailingCases.BOOL2BOOL_3_1_1_1_1 ON OPCUAServer.FailingServer.BOOL2BOOL_3_1_1_1_1;
    OpcUaBothFailingCases.SUBSCRIBE_NoObject_1 ON OPCUAServer.FailingServer.SUBSCRIBE_NoObject_1;
    OpcUaBothFailingCases.BOOL2BOOL_3_1_1_1_1_1 ON OPCUAServer.FailingServer.BOOL2BOOL_3_1_1_1_1_1;
    OpcUaBothFailingCases.SUBSCRIBE_NoObject ON OPCUAServer.FailingServer.SUBSCRIBE_NoObject;
    OpcUaBothFailingCases.BrowseWihtouObject ON OPCUAServer.FailingServer.BrowseWihtouObject;
    OpcUaBothFailingCases.wrongNamespace1 ON OPCUAServer.FailingServer.wrongNamespace1;
    OpcUaBothFailingCases.STRING2STRING_2 ON OPCUAServer.FailingServer.STRING2STRING_2;
    OpcUaBothFailingCases.Timeoutmethod ON OPCUAServer.FailingServer.Timeoutmethod;
    OpcUaBothFailingCases.E_DELAY_1 ON OPCUAServer.FailingServer.E_DELAY_1;
    OpcUaBothFailingCases.WrongInputOutput_1 ON OPCUACLient.FailingClient.WrongInputOutput_1;
    OpcUADelayedWorking.LocaMethods ON OPCUAServer.delayedWorkingServer.LocaMethods;
    OpcUADelayedWorking.E_SR ON OPCUAServer.delayedWorkingServer.E_SR;
    OpcUADelayedWorking.SUBSCRIBE_0_1 ON OPCUAServer.delayedWorkingServer.SUBSCRIBE_0_1;
    OpcUADelayedWorking.HandleInitLocal ON OPCUAServer.delayedWorkingServer.HandleInitLocal;
    OpcUADelayedWorking.E_PERMIT ON OPCUACLient.delayedWorkingClient.E_PERMIT;
    OpcUADelayedWorking.numericNodeIdTestRemote ON OPCUACLient.delayedWorkingClient.numericNodeIdTestRemote;
    OpcUADelayedWorking.RemoteMethods ON OPCUACLient.delayedWorkingClient.RemoteMethods;
    OpcUADelayedWorking.HandleInit ON OPCUACLient.delayedWorkingClient.HandleInit;
    OpcUADelayedWorking.PUBLISH_0 ON OPCUACLient.delayedWorkingClient.PUBLISH_0;
    OpcUADelayedWorking.InitFinishedSignal ON OPCUACLient.delayedWorkingClient.InitFinishedSignal;
    OpcUADelayedWorking.bytestringNodeIdTestRemote ON OPCUACLient.delayedWorkingClient.bytestringNodeIdTestRemote;
    OpcUADelayedWorking.E_DELAY ON OPCUACLient.delayedWorkingClient.E_DELAY;
    OpcUADelayedWorking.stringNodeIdTestRemote ON OPCUACLient.delayedWorkingClient.stringNodeIdTestRemote;
    OpcUADelayedWorking.E_SR_1 ON OPCUACLient.delayedWorkingClient.E_SR_1;
    OpcUADelayedWorking.E_SR_2 ON OPCUACLient.delayedWorkingClient.E_SR_2;
    OpcUADelayedWorking.folderTestRemote ON OPCUACLient.delayedWorkingClient.folderTestRemote;
    OpcUADelayedWorking.E_SWITCH ON OPCUAServer.delayedWorkingServer.E_SWITCH;
    OpcUADelayedWorking.E_DELAY_1 ON OPCUAServer.delayedWorkingServer.E_DELAY_1;
    OpcUADelayedWorking.E_SPLIT ON OPCUAServer.delayedWorkingServer.E_SPLIT;
    OpcUADelayedWorking.E_DELAY_1_1 ON OPCUAServer.delayedWorkingServer.E_DELAY_1_1;
    OpcUADelayedWorking.F_NOT ON OPCUAServer.delayedWorkingServer.F_NOT;
    OpcUADelayedWorking.E_PERMIT_1 ON OPCUAServer.delayedWorkingServer.E_PERMIT_1;
    OpcUaTypes.AllTypes ON OPCUAServer.typesServer.AllTypes;
    OpcUaTypes.LocalWrite ON OPCUAServer.typesServer.LocalWrite;
    OpcUaTypes.Method ON OPCUAServer.typesServer.Method;
    OpcUaTypes.TypeTest ON OPCUAServer.typesServer.TypeTest;
    OpcUaTypes.AllTypes_1 ON OPCUAServer.typesServer.AllTypes_1;
    OpcUaTypes.Read ON OPCUAServer.typesServer.Read;
    OpcUaTypes.TypeTest_1 ON OPCUAServer.typesServer.TypeTest_1;
    OpcUaTypes.E_SR ON OPCUAServer.typesServer.E_SR;
    OpcUaTypes.HandleInitLocal ON OPCUAServer.typesServer.HandleInitLocal;
    OpcUaTypes.SUBSCRIBE_0_1 ON OPCUAServer.typesServer.SUBSCRIBE_0_1;
    OpcUaTypes.E_SWITCH ON OPCUAServer.typesServer.E_SWITCH;
    OpcUaTypes.E_DELAY ON OPCUAServer.typesServer.E_DELAY;
    OpcUaTypes.SubApp_1 ON OPCUAServer.typesServer.SubApp_1;
    OpcUaTypes.SubApp_2 ON OPCUACLient.typesClient.SubApp_2;
    OpcUaTypes.RemoteRead ON OPCUACLient.typesClient.RemoteRead;
    OpcUaTypes.TypeTest_3 ON OPCUACLient.typesClient.TypeTest_3;
    OpcUaTypes.AllTypes_2 ON OPCUACLient.typesClient.AllTypes_2;
    OpcUaTypes.RemoteCall ON OPCUACLient.typesClient.RemoteCall;
    OpcUaTypes.AllTypes_3 ON OPCUACLient.typesClient.AllTypes_3;
    OpcUaTypes.TypeTest_2 ON OPCUACLient.typesClient.TypeTest_2;
    OpcUaTypes.HandleInit ON OPCUACLient.typesClient.HandleInit;
    OpcUaTypes.E_SR_1 ON OPCUACLient.typesClient.E_SR_1;
    OpcUaTypes.InitFinishedSignal ON OPCUACLient.typesClient.InitFinishedSignal;
    OpcUaTypes.E_PERMIT ON OPCUACLient.typesClient.E_PERMIT;
    OpcUaTypes.SubApp ON OPCUACLient.typesClient.SubApp;
    OpcUaTypes.E_SR_2 ON OPCUACLient.typesClient.E_SR_2;
    OpcUaTypes.PUBLISH_0 ON OPCUACLient.typesClient.PUBLISH_0;
    OpcUaBothWorking.stringNodeIdTest ON OPCUAServer.WorkingServer.stringNodeIdTest;
    OpcUaBothWorking.byteStringNodeIdTest ON OPCUAServer.WorkingServer.byteStringNodeIdTest;
    OpcUaBothWorking.numericNodeIdTest ON OPCUAServer.WorkingServer.numericNodeIdTest;
    OpcUADelayedWorking.numericNodeIdTest ON OPCUAServer.delayedWorkingServer.numericNodeIdTest;
    OpcUADelayedWorking.folderTest ON OPCUAServer.delayedWorkingServer.folderTest;
    OpcUADelayedWorking.byteStringNodeIdTest ON OPCUAServer.delayedWorkingServer.byteStringNodeIdTest;
    OpcUADelayedWorking.stringNodeIdTestt ON OPCUAServer.delayedWorkingServer.stringNodeIdTestt;
    OpcUaBothWorking.IsolatedCases ON OPCUAServer.WorkingServer.IsolatedCases;
    OpcUaBothWorking.RemoteIsolatedCases ON OPCUACLient.WorkingClient.RemoteIsolatedCases;
    OpcUaBothFailingCases.DINT2DINT_1_2 ON OPCUAServer.FailingServer.DINT2DINT_1_2;
    OpcUaBothFailingCases.PUBLISH_1 ON OPCUAServer.FailingServer.PUBLISH_1;
    ShortTests.DINT2DINT_1 ON OPCUAServer.TestServer.DINT2DINT_1;
    ShortTests.PUBLISH_1 ON OPCUAServer.TestServer.PUBLISH_1;
    ShortTests.PUBLISH_1_1 ON OPCUACLient.testClient.PUBLISH_1_1;
    ShortTests.DINT2DINT ON OPCUACLient.testClient.DINT2DINT;
    ShortTests.SUBSCRIBE_1 ON OPCUAServer.TestServer.SUBSCRIBE_1;
    ShortTests.DINT2DINT_1_1 ON OPCUAServer.TestServer.DINT2DINT_1_1;
    OpcUaBothFailingCases.SERVER_0_3 ON OPCUAServer.FailingServer.SERVER_0_3;
    OpcUaBothFailingCases.ObjectsFolder ON OPCUAServer.FailingServer.ObjectsFolder;
    OpcUaBothFailingCases.F_NOT_1_2_1_2_1_1 ON OPCUAServer.FailingServer.F_NOT_1_2_1_2_1_1;
    ShortTests.F_NOT_1_2_1_2_1_1 ON OPCUAServer.TestServer.F_NOT_1_2_1_2_1_1;
    ShortTests.ObjectsFolder ON OPCUAServer.TestServer.ObjectsFolder;
    ShortTests.SERVER_0_3 ON OPCUAServer.TestServer.SERVER_0_3;
    ShortTests.PUBLISH_1_1_1 ON OPCUAServer.TestServer.PUBLISH_1_1_1;
    ShortTests.SERVER_0 ON OPCUAServer.TestServer.SERVER_0;
    ShortTests.DINT2DINT_1_1_1 ON OPCUAServer.TestServer.DINT2DINT_1_1_1;
    OpcUaBothFailingCases.SERVER_0_4 ON OPCUAServer.FailingServer.SERVER_0_4;
    OpcUaTypes.RemoteWrite ON OPCUACLient.typesClient.RemoteWrite;
    OpcUaTypes.RemoteWriteAll ON OPCUACLient.typesClient.RemoteWriteAll;
    OpcUaBothWorking.WorkingWithoutSubscription ON OPCUACLient.WokingClientWithoutSubs.WorkingWithoutSubscription;
  END_MAPPINGS
  SEGMENTS
    Ethernet : Ethernet;
  END_SEGMENTS
  LINKS
    OPCUAServer => Ethernet;
    OPCUACLient => Ethernet;
  END_LINKS
END_SYSTEM
